EventTableTriggerIO 10058: Operator=0, IOValue=[1], IRC5Controller=? -1, SignalSource=SimulationProject 3637
EventTableTriggerIO 10059: Operator=0, IOValue=[0], IRC5Controller=? -1, SignalSource=SimulationProject 3637
EventTableTriggerIO 10060: Operator=0, IOValue=[0], IRC5Controller=? -1, SignalSource=SimulationProject 3637
EventTableTriggerIO 10061: Operator=0, IOValue=[0], IRC5Controller=? -1, SignalSource=SimulationProject 3637
EventTableTriggerIO 10062: Operator=0, IOValue=[1], IRC5Controller=? -1, SignalSource=SimulationProject 3637
EventTableTriggerIO 10063: Operator=0, IOValue=[1], IRC5Controller=? -1, SignalSource=SimulationProject 3637
EventTableTriggerIO 10064: Operator=0, IOValue=[1], IRC5Controller=? -1, SignalSource=SimulationProject 3637
EventTableTriggerIO 10065: Operator=0, IOValue=[0], IRC5Controller=? -1, SignalSource=SimulationProject 3637
EventTableTriggerIO 10066: Operator=0, IOValue=[0], IRC5Controller=? -1, SignalSource=SimulationProject 3637
EventTableTriggerIO 10067: Operator=0, IOValue=[0], IRC5Controller=? -1, SignalSource=SimulationProject 3637
EventTableTriggerIO 10068: Operator=0, IOValue=[1], IRC5Controller=? -1, SignalSource=SimulationProject 3637
EventTableTriggerIO 10069: Operator=0, IOValue=[1], IRC5Controller=? -1, SignalSource=SimulationProject 3637
EventTableTriggerIO 10070: Operator=0, IOValue=[1], IRC5Controller=? -1, SignalSource=SimulationProject 3637
EventTableTriggerIO 10071: Operator=0, IOValue=[0], IRC5Controller=? -1, SignalSource=SimulationProject 3637
EventTableTriggerIO 10072: Operator=0, IOValue=[0], IRC5Controller=? -1, SignalSource=SimulationProject 3637
EventTableTriggerIO 10073: Operator=0, IOValue=[0], IRC5Controller=? -1, SignalSource=SimulationProject 3637
EventTableTriggerIO 10074: Operator=0, IOValue=[1], IRC5Controller=? -1, SignalSource=SimulationProject 3637
EventTableTriggerIO 10075: Operator=0, IOValue=[1], IRC5Controller=? -1, SignalSource=SimulationProject 3637
EventTableTriggerIO 10076: Operator=0, IOValue=[1], IRC5Controller=? -1, SignalSource=SimulationProject 3637
EventTableTriggerIO 10077: Operator=0, IOValue=[0], IRC5Controller=? -1, SignalSource=SimulationProject 3637
EventTableTriggerIO 10078: Operator=0, IOValue=[0], IRC5Controller=? -1, SignalSource=SimulationProject 3637
EventTableTriggerIO 10079: Operator=0, IOValue=[0], IRC5Controller=? -1, SignalSource=SimulationProject 3637
EventTableTriggerIO 10087: Operator=0, IOValue=[1], IRC5Controller=? -1, SignalSource=SimulationProject 3637
EventTableTriggerIO 10088: Operator=0, IOValue=[0], IRC5Controller=? -1, SignalSource=SimulationProject 3637
EventTableTriggerIO 10089: Operator=0, IOValue=[1], IRC5Controller=? -1, SignalSource=SimulationProject 3637
EventTableTriggerIO 10090: Operator=0, IOValue=[0], IRC5Controller=? -1, SignalSource=SimulationProject 3637
EventTableTriggerIO 10091: Operator=0, IOValue=[1], IRC5Controller=? -1, SignalSource=SimulationProject 3637
EventTableTriggerIO 10092: Operator=0, IOValue=[0], IRC5Controller=? -1, SignalSource=SimulationProject 3637
EventTableTriggerIO 10093: Operator=0, IOValue=[1], IRC5Controller=? -1, SignalSource=SimulationProject 3637
EventTableTriggerIO 10094: Operator=0, IOValue=[0], IRC5Controller=? -1, SignalSource=SimulationProject 3637
EventTableTriggerIO 10095: Operator=0, IOValue=[1], IRC5Controller=? -1, SignalSource=SimulationProject 3637
EventTableTriggerIO 10096: Operator=0, IOValue=[0], IRC5Controller=? -1, SignalSource=SimulationProject 3637
EventTableTriggerIO 10097: Operator=0, IOValue=[1], IRC5Controller=? -1, SignalSource=SimulationProject 3637
EventTableTriggerIO 10098: Operator=0, IOValue=[0], IRC5Controller=? -1, SignalSource=SimulationProject 3637
EventTableTriggerIO 10099: Operator=0, IOValue=[1], IRC5Controller=? -1, SignalSource=SimulationProject 3637
EventTableTriggerIO 10100: Operator=0, IOValue=[0], IRC5Controller=? -1, SignalSource=SimulationProject 3637
EventTableTriggerIO 10101: Operator=0, IOValue=[1], IRC5Controller=? -1, SignalSource=SimulationProject 3637
EventTableTriggerIO 10102: Operator=0, IOValue=[0], IRC5Controller=? -1, SignalSource=SimulationProject 3637
EventTableTriggerIO 10103: Operator=0, IOValue=[1], IRC5Controller=? -1, SignalSource=SimulationProject 3637
EventTableTriggerIO 10104: Operator=0, IOValue=[0], IRC5Controller=? -1, SignalSource=SimulationProject 3637
EventTableTriggerIO 10105: Operator=0, IOValue=[1], IRC5Controller=? -1, SignalSource=SimulationProject 3637
EventTableTriggerIO 10106: Operator=0, IOValue=[0], IRC5Controller=? -1, SignalSource=SimulationProject 3637
EventTableTriggerIO 10107: Operator=0, IOValue=[1], IRC5Controller=? -1, SignalSource=SimulationProject 3637
EventTableTriggerIO 10108: Operator=0, IOValue=[0], IRC5Controller=? -1, SignalSource=SimulationProject 3637
EventTableTriggerIO 10109: Operator=0, IOValue=[1], IRC5Controller=? -1, SignalSource=SimulationProject 3637
EventTableTriggerIO 10110: Operator=0, IOValue=[0], IRC5Controller=? -1, SignalSource=SimulationProject 3637
EventTableTriggerIO 10194: Operator=0, IOValue=[1], IRC5Controller=? -1, SignalSource=SimulationProject 3637
EventTableTriggerIO 10195: Operator=0, IOValue=[1], IRC5Controller=? -1, SignalSource=SimulationProject 3637
EventTableTriggerIO 10196: Operator=0, IOValue=[0], IRC5Controller=? -1, SignalSource=SimulationProject 3637
EventTableTriggerIO 10197: Operator=0, IOValue=[0], IRC5Controller=? -1, SignalSource=SimulationProject 3637
EventTableTriggerIO 10198: Operator=0, IOValue=[1], IRC5Controller=? -1, SignalSource=SimulationProject 3637
EventTableTriggerIO 10199: Operator=0, IOValue=[1], IRC5Controller=? -1, SignalSource=SimulationProject 3637
EventTableTriggerIO 10200: Operator=0, IOValue=[0], IRC5Controller=? -1, SignalSource=SimulationProject 3637
EventTableTriggerIO 10201: Operator=0, IOValue=[0], IRC5Controller=? -1, SignalSource=SimulationProject 3637
EventTableTriggerIO 10202: Operator=0, IOValue=[1], IRC5Controller=? -1, SignalSource=SimulationProject 3637
EventTableTriggerIO 10203: Operator=0, IOValue=[1], IRC5Controller=? -1, SignalSource=SimulationProject 3637
EventTableTriggerIO 10204: Operator=0, IOValue=[0], IRC5Controller=? -1, SignalSource=SimulationProject 3637
EventTableTriggerIO 10205: Operator=0, IOValue=[0], IRC5Controller=? -1, SignalSource=SimulationProject 3637
EventTableTriggerIO 10206: Operator=0, IOValue=[1], IRC5Controller=? -1, SignalSource=SimulationProject 3637
EventTableTriggerIO 10207: Operator=0, IOValue=[1], IRC5Controller=? -1, SignalSource=SimulationProject 3637
EventTableTriggerIO 10208: Operator=0, IOValue=[0], IRC5Controller=? -1, SignalSource=SimulationProject 3637
EventTableTriggerIO 10209: Operator=0, IOValue=[0], IRC5Controller=? -1, SignalSource=SimulationProject 3637
EventTableTriggerIO 10210: Operator=0, IOValue=[1], IRC5Controller=? -1, SignalSource=SimulationProject 3637
EventTableTriggerIO 10211: Operator=0, IOValue=[1], IRC5Controller=? -1, SignalSource=SimulationProject 3637
EventTableTriggerIO 10212: Operator=0, IOValue=[0], IRC5Controller=? -1, SignalSource=SimulationProject 3637
EventTableTriggerIO 10213: Operator=0, IOValue=[0], IRC5Controller=? -1, SignalSource=SimulationProject 3637
EventTableTriggerIO 10214: Operator=0, IOValue=[1], IRC5Controller=? -1, SignalSource=SimulationProject 3637
EventTableTriggerIO 10215: Operator=0, IOValue=[1], IRC5Controller=? -1, SignalSource=SimulationProject 3637
EventTableTriggerIO 10216: Operator=0, IOValue=[0], IRC5Controller=? -1, SignalSource=SimulationProject 3637
EventTableTriggerIO 10217: Operator=0, IOValue=[0], IRC5Controller=? -1, SignalSource=SimulationProject 3637
EventTableTriggerIO 10218: Operator=0, IOValue=[1], IRC5Controller=? -1, SignalSource=SimulationProject 3637
EventTableTriggerIO 10219: Operator=0, IOValue=[1], IRC5Controller=? -1, SignalSource=SimulationProject 3637
EventTableTriggerIO 10220: Operator=0, IOValue=[0], IRC5Controller=? -1, SignalSource=SimulationProject 3637
EventTableTriggerIO 10221: Operator=0, IOValue=[0], IRC5Controller=? -1, SignalSource=SimulationProject 3637
EventTableTriggerIO 10222: Operator=0, IOValue=[1], IRC5Controller=? -1, SignalSource=SimulationProject 3637
EventTableTriggerIO 10223: Operator=0, IOValue=[1], IRC5Controller=? -1, SignalSource=SimulationProject 3637
EventTableTriggerIO 10224: Operator=0, IOValue=[0], IRC5Controller=? -1, SignalSource=SimulationProject 3637
EventTableTriggerIO 10225: Operator=0, IOValue=[0], IRC5Controller=? -1, SignalSource=SimulationProject 3637
EventTableTriggerIO 10226: Operator=0, IOValue=[1], IRC5Controller=? -1, SignalSource=SimulationProject 3637
EventTableTriggerIO 10227: Operator=0, IOValue=[1], IRC5Controller=? -1, SignalSource=SimulationProject 3637
EventTableTriggerIO 10228: Operator=0, IOValue=[0], IRC5Controller=? -1, SignalSource=SimulationProject 3637
EventTableTriggerIO 10229: Operator=0, IOValue=[0], IRC5Controller=? -1, SignalSource=SimulationProject 3637
EventTableTriggerIO 10230: Operator=0, IOValue=[1], IRC5Controller=? -1, SignalSource=SimulationProject 3637
EventTableTriggerIO 10231: Operator=0, IOValue=[1], IRC5Controller=? -1, SignalSource=SimulationProject 3637
EventTableTriggerIO 10232: Operator=0, IOValue=[0], IRC5Controller=? -1, SignalSource=SimulationProject 3637
EventTableTriggerIO 10233: Operator=0, IOValue=[0], IRC5Controller=? -1, SignalSource=SimulationProject 3637
EventTableTriggerIO 10234: Operator=0, IOValue=[1], IRC5Controller=? -1, SignalSource=SimulationProject 3637
EventTableTriggerIO 10235: Operator=0, IOValue=[1], IRC5Controller=? -1, SignalSource=SimulationProject 3637
EventTableTriggerIO 10236: Operator=0, IOValue=[0], IRC5Controller=? -1, SignalSource=SimulationProject 3637
EventTableTriggerIO 10237: Operator=0, IOValue=[0], IRC5Controller=? -1, SignalSource=SimulationProject 3637
EventTableTriggerIO 10238: Operator=0, IOValue=[1], IRC5Controller=? -1, SignalSource=SimulationProject 3637
EventTableTriggerIO 10239: Operator=0, IOValue=[1], IRC5Controller=? -1, SignalSource=SimulationProject 3637
EventTableTriggerIO 10240: Operator=0, IOValue=[0], IRC5Controller=? -1, SignalSource=SimulationProject 3637
EventTableTriggerIO 10241: Operator=0, IOValue=[0], IRC5Controller=? -1, SignalSource=SimulationProject 3637
EventTableEntry 10242: ActivationMode=2, Cyclic=false, Group=, Trigger=doAxelTool_L 10243, Actions=[EventTableActionAttach 10244], Comment=
EventTableTriggerIO 10243: Operator=0, IOValue=[1], IRC5Controller=? -1, SignalSource=SimulationProject 3637
EventTableActionAttach 10244: MountObject=false, FlangeIndext=0, FindNearest=false, AttachmentParent=IRB6660_100_335__01_L 3595, AttachmentChild=AxelPinTool_L 5996, Offset=[X=1, Y=0, Z=0, W=0, X=0, Y=1, Z=0, W=0, X=0, Y=0, Z=1, W=0, X=0, Y=0, Z=0, W=1]
EventTableTriggerIO 10245: Operator=0, IOValue=[1], IRC5Controller=? -1, SignalSource=SimulationProject 3637
EventTableEntry 10246: ActivationMode=2, Cyclic=false, Group=, Trigger=doAxelTool_L 10247, Actions=[EventTableActionDetach 10248], Comment=
EventTableTriggerIO 10247: Operator=0, IOValue=[0], IRC5Controller=? -1, SignalSource=SimulationProject 3637
EventTableActionDetach 10248: AttachmentParent=IRB6660_100_335__01_L 3595, AttachmentChild=AxelPinTool_L 5996
EventTableTriggerIO 10249: Operator=0, IOValue=[0], IRC5Controller=? -1, SignalSource=SimulationProject 3637
EventTableEntry 10250: ActivationMode=2, Cyclic=false, Group=, Trigger=doAxel_L 10251, Actions=[EventTableActionAttach 10252], Comment=
EventTableTriggerIO 10251: Operator=0, IOValue=[1], IRC5Controller=? -1, SignalSource=SimulationProject 3637
EventTableActionAttach 10252: MountObject=false, FlangeIndext=0, FindNearest=true, AttachmentParent=AxelPinTool_L 5996, AttachmentChild=? -1, Offset=[X=1, Y=0, Z=0, W=0, X=0, Y=1, Z=0, W=0, X=0, Y=0, Z=1, W=0, X=0, Y=0, Z=0, W=1]
EventTableTriggerIO 10253: Operator=0, IOValue=[1], IRC5Controller=? -1, SignalSource=SimulationProject 3637
EventTableEntry 10254: ActivationMode=2, Cyclic=false, Group=, Trigger=doAxel_L 10255, Actions=[EventTableActionDetach 10256], Comment=
EventTableTriggerIO 10255: Operator=0, IOValue=[0], IRC5Controller=? -1, SignalSource=SimulationProject 3637
EventTableActionDetach 10256: AttachmentParent=AxelPinTool_L 5996, AttachmentChild=? -1
EventTableTriggerIO 10257: Operator=0, IOValue=[0], IRC5Controller=? -1, SignalSource=SimulationProject 3637
EventTableTriggerIO 10629: Operator=0, IOValue=[1], IRC5Controller=? -1, SignalSource=SimulationProject 3637
EventTableTriggerIO 10630: Operator=0, IOValue=[0], IRC5Controller=? -1, SignalSource=SimulationProject 3637
EventTableTriggerIO 10631: Operator=0, IOValue=[1], IRC5Controller=? -1, SignalSource=SimulationProject 3637
EventTableTriggerIO 10632: Operator=0, IOValue=[0], IRC5Controller=? -1, SignalSource=SimulationProject 3637
EventTableTriggerIO 10633: Operator=0, IOValue=[1], IRC5Controller=? -1, SignalSource=SimulationProject 3637
EventTableTriggerIO 10634: Operator=0, IOValue=[0], IRC5Controller=? -1, SignalSource=SimulationProject 3637
EventTableTriggerIO 10635: Operator=0, IOValue=[1], IRC5Controller=? -1, SignalSource=SimulationProject 3637
EventTableTriggerIO 10636: Operator=0, IOValue=[0], IRC5Controller=? -1, SignalSource=SimulationProject 3637
EventTableTriggerIO 10637: Operator=0, IOValue=[1], IRC5Controller=? -1, SignalSource=SimulationProject 3637
EventTableTriggerIO 10638: Operator=0, IOValue=[0], IRC5Controller=? -1, SignalSource=SimulationProject 3637
EventTableTriggerIO 10639: Operator=0, IOValue=[1], IRC5Controller=? -1, SignalSource=SimulationProject 3637
EventTableTriggerIO 10640: Operator=0, IOValue=[0], IRC5Controller=? -1, SignalSource=SimulationProject 3637
EventTableTriggerIO 10641: Operator=0, IOValue=[1], IRC5Controller=? -1, SignalSource=SimulationProject 3637
EventTableTriggerIO 10642: Operator=0, IOValue=[0], IRC5Controller=? -1, SignalSource=SimulationProject 3637
EventTableTriggerIO 10643: Operator=0, IOValue=[1], IRC5Controller=? -1, SignalSource=SimulationProject 3637
EventTableTriggerIO 10644: Operator=0, IOValue=[0], IRC5Controller=? -1, SignalSource=SimulationProject 3637
EventTableTriggerIO 10645: Operator=0, IOValue=[1], IRC5Controller=? -1, SignalSource=SimulationProject 3637
EventTableTriggerIO 10646: Operator=0, IOValue=[0], IRC5Controller=? -1, SignalSource=SimulationProject 3637
EventTableTriggerIO 10647: Operator=0, IOValue=[1], IRC5Controller=? -1, SignalSource=SimulationProject 3637
EventTableTriggerIO 10648: Operator=0, IOValue=[0], IRC5Controller=? -1, SignalSource=SimulationProject 3637
EventTableTriggerIO 10649: Operator=0, IOValue=[1], IRC5Controller=? -1, SignalSource=SimulationProject 3637
EventTableTriggerIO 10650: Operator=0, IOValue=[0], IRC5Controller=? -1, SignalSource=SimulationProject 3637
EventTableTriggerIO 10651: Operator=0, IOValue=[1], IRC5Controller=? -1, SignalSource=SimulationProject 3637
EventTableTriggerIO 10652: Operator=0, IOValue=[0], IRC5Controller=? -1, SignalSource=SimulationProject 3637
EventTableTriggerIO 10653: Operator=0, IOValue=[1], IRC5Controller=? -1, SignalSource=SimulationProject 3637
EventTableTriggerIO 10654: Operator=0, IOValue=[0], IRC5Controller=? -1, SignalSource=SimulationProject 3637
EventTableTriggerIO 10655: Operator=0, IOValue=[1], IRC5Controller=? -1, SignalSource=SimulationProject 3637
EventTableTriggerIO 10656: Operator=0, IOValue=[0], IRC5Controller=? -1, SignalSource=SimulationProject 3637
EventTableTriggerIO 10664: Operator=0, IOValue=[1], IRC5Controller=? -1, SignalSource=SimulationProject 3637
EventTableTriggerIO 10665: Operator=0, IOValue=[0], IRC5Controller=? -1, SignalSource=SimulationProject 3637
EventTableTriggerIO 10666: Operator=0, IOValue=[1], IRC5Controller=? -1, SignalSource=SimulationProject 3637
EventTableTriggerIO 10667: Operator=0, IOValue=[0], IRC5Controller=? -1, SignalSource=SimulationProject 3637
EventTableTriggerIO 10668: Operator=0, IOValue=[1], IRC5Controller=? -1, SignalSource=SimulationProject 3637
EventTableTriggerIO 10669: Operator=0, IOValue=[0], IRC5Controller=? -1, SignalSource=SimulationProject 3637
EventTableTriggerIO 10670: Operator=0, IOValue=[1], IRC5Controller=? -1, SignalSource=SimulationProject 3637
EventTableTriggerIO 10671: Operator=0, IOValue=[0], IRC5Controller=? -1, SignalSource=SimulationProject 3637
EventTableTriggerIO 10672: Operator=0, IOValue=[1], IRC5Controller=? -1, SignalSource=SimulationProject 3637
EventTableTriggerIO 10673: Operator=0, IOValue=[0], IRC5Controller=? -1, SignalSource=SimulationProject 3637
EventTableTriggerIO 10674: Operator=0, IOValue=[1], IRC5Controller=? -1, SignalSource=SimulationProject 3637
EventTableTriggerIO 10675: Operator=0, IOValue=[0], IRC5Controller=? -1, SignalSource=SimulationProject 3637
EventTableTriggerIO 10676: Operator=0, IOValue=[1], IRC5Controller=? -1, SignalSource=SimulationProject 3637
EventTableTriggerIO 10677: Operator=0, IOValue=[0], IRC5Controller=? -1, SignalSource=SimulationProject 3637
EventTableTriggerIO 10678: Operator=0, IOValue=[1], IRC5Controller=? -1, SignalSource=SimulationProject 3637
EventTableTriggerIO 10679: Operator=0, IOValue=[0], IRC5Controller=? -1, SignalSource=SimulationProject 3637
EventTableTriggerIO 10680: Operator=0, IOValue=[1], IRC5Controller=? -1, SignalSource=SimulationProject 3637
EventTableTriggerIO 10681: Operator=0, IOValue=[0], IRC5Controller=? -1, SignalSource=SimulationProject 3637
EventTableTriggerIO 10682: Operator=0, IOValue=[1], IRC5Controller=? -1, SignalSource=SimulationProject 3637
EventTableTriggerIO 10683: Operator=0, IOValue=[0], IRC5Controller=? -1, SignalSource=SimulationProject 3637
EventTableTriggerIO 10684: Operator=0, IOValue=[1], IRC5Controller=? -1, SignalSource=SimulationProject 3637
EventTableTriggerIO 10685: Operator=0, IOValue=[0], IRC5Controller=? -1, SignalSource=SimulationProject 3637
EventTableTriggerIO 10686: Operator=0, IOValue=[1], IRC5Controller=? -1, SignalSource=SimulationProject 3637
EventTableTriggerIO 10687: Operator=0, IOValue=[0], IRC5Controller=? -1, SignalSource=SimulationProject 3637
EventTableTriggerIO 10688: Operator=0, IOValue=[1], IRC5Controller=? -1, SignalSource=SimulationProject 3637
EventTableTriggerIO 10689: Operator=0, IOValue=[0], IRC5Controller=? -1, SignalSource=SimulationProject 3637
EventTableTriggerIO 10690: Operator=0, IOValue=[1], IRC5Controller=? -1, SignalSource=SimulationProject 3637
EventTableTriggerIO 10691: Operator=0, IOValue=[0], IRC5Controller=? -1, SignalSource=SimulationProject 3637
EventTableTriggerIO 10748: Operator=0, IOValue=[1], IRC5Controller=? -1, SignalSource=SimulationProject 3637
EventTableTriggerIO 10749: Operator=0, IOValue=[1], IRC5Controller=? -1, SignalSource=SimulationProject 3637
EventTableTriggerIO 10750: Operator=0, IOValue=[1], IRC5Controller=? -1, SignalSource=SimulationProject 3637
EventTableTriggerIO 10751: Operator=0, IOValue=[0], IRC5Controller=? -1, SignalSource=SimulationProject 3637
EventTableTriggerIO 10752: Operator=0, IOValue=[0], IRC5Controller=? -1, SignalSource=SimulationProject 3637
EventTableTriggerIO 10753: Operator=0, IOValue=[0], IRC5Controller=? -1, SignalSource=SimulationProject 3637
EventTableTriggerIO 10754: Operator=0, IOValue=[1], IRC5Controller=? -1, SignalSource=SimulationProject 3637
EventTableTriggerIO 10755: Operator=0, IOValue=[1], IRC5Controller=? -1, SignalSource=SimulationProject 3637
EventTableTriggerIO 10756: Operator=0, IOValue=[1], IRC5Controller=? -1, SignalSource=SimulationProject 3637
EventTableTriggerIO 10757: Operator=0, IOValue=[0], IRC5Controller=? -1, SignalSource=SimulationProject 3637
EventTableTriggerIO 10758: Operator=0, IOValue=[0], IRC5Controller=? -1, SignalSource=SimulationProject 3637
EventTableTriggerIO 10759: Operator=0, IOValue=[0], IRC5Controller=? -1, SignalSource=SimulationProject 3637
EventTableTriggerIO 10760: Operator=0, IOValue=[1], IRC5Controller=? -1, SignalSource=SimulationProject 3637
EventTableTriggerIO 10761: Operator=0, IOValue=[1], IRC5Controller=? -1, SignalSource=SimulationProject 3637
EventTableTriggerIO 10762: Operator=0, IOValue=[1], IRC5Controller=? -1, SignalSource=SimulationProject 3637
EventTableTriggerIO 10763: Operator=0, IOValue=[0], IRC5Controller=? -1, SignalSource=SimulationProject 3637
EventTableTriggerIO 10764: Operator=0, IOValue=[0], IRC5Controller=? -1, SignalSource=SimulationProject 3637
EventTableTriggerIO 10765: Operator=0, IOValue=[0], IRC5Controller=? -1, SignalSource=SimulationProject 3637
EventTableTriggerIO 10766: Operator=0, IOValue=[1], IRC5Controller=? -1, SignalSource=SimulationProject 3637
EventTableTriggerIO 10767: Operator=0, IOValue=[1], IRC5Controller=? -1, SignalSource=SimulationProject 3637
EventTableTriggerIO 10768: Operator=0, IOValue=[1], IRC5Controller=? -1, SignalSource=SimulationProject 3637
EventTableTriggerIO 10769: Operator=0, IOValue=[0], IRC5Controller=? -1, SignalSource=SimulationProject 3637
EventTableTriggerIO 10770: Operator=0, IOValue=[0], IRC5Controller=? -1, SignalSource=SimulationProject 3637
EventTableTriggerIO 10771: Operator=0, IOValue=[0], IRC5Controller=? -1, SignalSource=SimulationProject 3637
EventTableTriggerIO 10772: Operator=0, IOValue=[1], IRC5Controller=? -1, SignalSource=SimulationProject 3637
EventTableTriggerIO 10773: Operator=0, IOValue=[1], IRC5Controller=? -1, SignalSource=SimulationProject 3637
EventTableTriggerIO 10774: Operator=0, IOValue=[1], IRC5Controller=? -1, SignalSource=SimulationProject 3637
EventTableTriggerIO 10775: Operator=0, IOValue=[0], IRC5Controller=? -1, SignalSource=SimulationProject 3637
EventTableTriggerIO 10776: Operator=0, IOValue=[0], IRC5Controller=? -1, SignalSource=SimulationProject 3637
EventTableTriggerIO 10777: Operator=0, IOValue=[0], IRC5Controller=? -1, SignalSource=SimulationProject 3637
EventTableTriggerIO 10778: Operator=0, IOValue=[1], IRC5Controller=? -1, SignalSource=SimulationProject 3637
EventTableTriggerIO 10779: Operator=0, IOValue=[1], IRC5Controller=? -1, SignalSource=SimulationProject 3637
EventTableTriggerIO 10780: Operator=0, IOValue=[1], IRC5Controller=? -1, SignalSource=SimulationProject 3637
EventTableTriggerIO 10781: Operator=0, IOValue=[0], IRC5Controller=? -1, SignalSource=SimulationProject 3637
EventTableTriggerIO 10782: Operator=0, IOValue=[0], IRC5Controller=? -1, SignalSource=SimulationProject 3637
EventTableTriggerIO 10783: Operator=0, IOValue=[0], IRC5Controller=? -1, SignalSource=SimulationProject 3637
EventTableTriggerIO 10784: Operator=0, IOValue=[1], IRC5Controller=? -1, SignalSource=SimulationProject 3637
EventTableTriggerIO 10785: Operator=0, IOValue=[1], IRC5Controller=? -1, SignalSource=SimulationProject 3637
EventTableTriggerIO 10786: Operator=0, IOValue=[1], IRC5Controller=? -1, SignalSource=SimulationProject 3637
EventTableTriggerIO 10787: Operator=0, IOValue=[0], IRC5Controller=? -1, SignalSource=SimulationProject 3637
EventTableTriggerIO 10788: Operator=0, IOValue=[0], IRC5Controller=? -1, SignalSource=SimulationProject 3637
EventTableTriggerIO 10789: Operator=0, IOValue=[0], IRC5Controller=? -1, SignalSource=SimulationProject 3637
EventTableTriggerIO 10790: Operator=0, IOValue=[1], IRC5Controller=? -1, SignalSource=SimulationProject 3637
EventTableTriggerIO 10791: Operator=0, IOValue=[1], IRC5Controller=? -1, SignalSource=SimulationProject 3637
EventTableTriggerIO 10792: Operator=0, IOValue=[1], IRC5Controller=? -1, SignalSource=SimulationProject 3637
EventTableTriggerIO 10793: Operator=0, IOValue=[0], IRC5Controller=? -1, SignalSource=SimulationProject 3637
EventTableTriggerIO 10794: Operator=0, IOValue=[0], IRC5Controller=? -1, SignalSource=SimulationProject 3637
EventTableTriggerIO 10795: Operator=0, IOValue=[0], IRC5Controller=? -1, SignalSource=SimulationProject 3637
EventTableTriggerIO 10796: Operator=0, IOValue=[1], IRC5Controller=? -1, SignalSource=SimulationProject 3637
EventTableTriggerIO 10797: Operator=0, IOValue=[1], IRC5Controller=? -1, SignalSource=SimulationProject 3637
EventTableTriggerIO 10798: Operator=0, IOValue=[1], IRC5Controller=? -1, SignalSource=SimulationProject 3637
EventTableTriggerIO 10799: Operator=0, IOValue=[0], IRC5Controller=? -1, SignalSource=SimulationProject 3637
EventTableTriggerIO 10800: Operator=0, IOValue=[0], IRC5Controller=? -1, SignalSource=SimulationProject 3637
EventTableTriggerIO 10801: Operator=0, IOValue=[0], IRC5Controller=? -1, SignalSource=SimulationProject 3637
EventTableTriggerIO 10802: Operator=0, IOValue=[1], IRC5Controller=? -1, SignalSource=SimulationProject 3637
EventTableTriggerIO 10803: Operator=0, IOValue=[1], IRC5Controller=? -1, SignalSource=SimulationProject 3637
EventTableTriggerIO 10804: Operator=0, IOValue=[1], IRC5Controller=? -1, SignalSource=SimulationProject 3637
EventTableTriggerIO 10805: Operator=0, IOValue=[0], IRC5Controller=? -1, SignalSource=SimulationProject 3637
EventTableTriggerIO 10806: Operator=0, IOValue=[0], IRC5Controller=? -1, SignalSource=SimulationProject 3637
EventTableTriggerIO 10807: Operator=0, IOValue=[0], IRC5Controller=? -1, SignalSource=SimulationProject 3637
EventTableTriggerIO 10808: Operator=0, IOValue=[1], IRC5Controller=? -1, SignalSource=SimulationProject 3637
EventTableTriggerIO 10809: Operator=0, IOValue=[1], IRC5Controller=? -1, SignalSource=SimulationProject 3637
EventTableTriggerIO 10810: Operator=0, IOValue=[1], IRC5Controller=? -1, SignalSource=SimulationProject 3637
EventTableTriggerIO 10811: Operator=0, IOValue=[0], IRC5Controller=? -1, SignalSource=SimulationProject 3637
EventTableTriggerIO 10812: Operator=0, IOValue=[0], IRC5Controller=? -1, SignalSource=SimulationProject 3637
EventTableTriggerIO 10813: Operator=0, IOValue=[0], IRC5Controller=? -1, SignalSource=SimulationProject 3637
EventTableTriggerIO 10814: Operator=0, IOValue=[1], IRC5Controller=? -1, SignalSource=SimulationProject 3637
EventTableTriggerIO 10815: Operator=0, IOValue=[1], IRC5Controller=? -1, SignalSource=SimulationProject 3637
EventTableTriggerIO 10816: Operator=0, IOValue=[1], IRC5Controller=? -1, SignalSource=SimulationProject 3637
EventTableTriggerIO 10817: Operator=0, IOValue=[0], IRC5Controller=? -1, SignalSource=SimulationProject 3637
EventTableTriggerIO 10818: Operator=0, IOValue=[0], IRC5Controller=? -1, SignalSource=SimulationProject 3637
EventTableTriggerIO 10819: Operator=0, IOValue=[0], IRC5Controller=? -1, SignalSource=SimulationProject 3637
EventTableTriggerIO 10820: Operator=0, IOValue=[1], IRC5Controller=? -1, SignalSource=SimulationProject 3637
EventTableTriggerIO 10821: Operator=0, IOValue=[1], IRC5Controller=? -1, SignalSource=SimulationProject 3637
EventTableTriggerIO 10822: Operator=0, IOValue=[1], IRC5Controller=? -1, SignalSource=SimulationProject 3637
EventTableTriggerIO 10823: Operator=0, IOValue=[0], IRC5Controller=? -1, SignalSource=SimulationProject 3637
EventTableTriggerIO 10824: Operator=0, IOValue=[0], IRC5Controller=? -1, SignalSource=SimulationProject 3637
EventTableTriggerIO 10825: Operator=0, IOValue=[0], IRC5Controller=? -1, SignalSource=SimulationProject 3637
EventTableTriggerIO 10826: Operator=0, IOValue=[1], IRC5Controller=? -1, SignalSource=SimulationProject 3637
EventTableTriggerIO 10827: Operator=0, IOValue=[1], IRC5Controller=? -1, SignalSource=SimulationProject 3637
EventTableTriggerIO 10828: Operator=0, IOValue=[1], IRC5Controller=? -1, SignalSource=SimulationProject 3637
EventTableTriggerIO 10829: Operator=0, IOValue=[0], IRC5Controller=? -1, SignalSource=SimulationProject 3637
EventTableTriggerIO 10830: Operator=0, IOValue=[0], IRC5Controller=? -1, SignalSource=SimulationProject 3637
EventTableTriggerIO 10831: Operator=0, IOValue=[0], IRC5Controller=? -1, SignalSource=SimulationProject 3637
EventTableTriggerIO 11467: Operator=0, IOValue=[1], IRC5Controller=? -1, SignalSource=SimulationProject 3637
EventTableTriggerIO 11468: Operator=0, IOValue=[1], IRC5Controller=? -1, SignalSource=SimulationProject 3637
EventTableTriggerIO 11469: Operator=0, IOValue=[0], IRC5Controller=? -1, SignalSource=SimulationProject 3637
EventTableTriggerIO 11470: Operator=0, IOValue=[0], IRC5Controller=? -1, SignalSource=SimulationProject 3637
EventTableTriggerIO 11471: Operator=0, IOValue=[1], IRC5Controller=? -1, SignalSource=SimulationProject 3637
EventTableTriggerIO 11472: Operator=0, IOValue=[1], IRC5Controller=? -1, SignalSource=SimulationProject 3637
EventTableTriggerIO 11473: Operator=0, IOValue=[0], IRC5Controller=? -1, SignalSource=SimulationProject 3637
EventTableTriggerIO 11474: Operator=0, IOValue=[0], IRC5Controller=? -1, SignalSource=SimulationProject 3637
EventTableTriggerIO 11475: Operator=0, IOValue=[1], IRC5Controller=? -1, SignalSource=SimulationProject 3637
EventTableTriggerIO 11476: Operator=0, IOValue=[1], IRC5Controller=? -1, SignalSource=SimulationProject 3637
EventTableTriggerIO 11477: Operator=0, IOValue=[0], IRC5Controller=? -1, SignalSource=SimulationProject 3637
EventTableTriggerIO 11478: Operator=0, IOValue=[0], IRC5Controller=? -1, SignalSource=SimulationProject 3637
EventTableTriggerIO 11479: Operator=0, IOValue=[1], IRC5Controller=? -1, SignalSource=SimulationProject 3637
EventTableTriggerIO 11480: Operator=0, IOValue=[1], IRC5Controller=? -1, SignalSource=SimulationProject 3637
EventTableTriggerIO 11481: Operator=0, IOValue=[0], IRC5Controller=? -1, SignalSource=SimulationProject 3637
EventTableTriggerIO 11482: Operator=0, IOValue=[0], IRC5Controller=? -1, SignalSource=SimulationProject 3637
EventTableTriggerIO 11483: Operator=0, IOValue=[1], IRC5Controller=? -1, SignalSource=SimulationProject 3637
EventTableTriggerIO 11484: Operator=0, IOValue=[1], IRC5Controller=? -1, SignalSource=SimulationProject 3637
EventTableTriggerIO 11485: Operator=0, IOValue=[0], IRC5Controller=? -1, SignalSource=SimulationProject 3637
EventTableTriggerIO 11486: Operator=0, IOValue=[0], IRC5Controller=? -1, SignalSource=SimulationProject 3637
EventTableTriggerIO 11487: Operator=0, IOValue=[1], IRC5Controller=? -1, SignalSource=SimulationProject 3637
EventTableTriggerIO 11488: Operator=0, IOValue=[1], IRC5Controller=? -1, SignalSource=SimulationProject 3637
EventTableTriggerIO 11489: Operator=0, IOValue=[0], IRC5Controller=? -1, SignalSource=SimulationProject 3637
EventTableTriggerIO 11490: Operator=0, IOValue=[0], IRC5Controller=? -1, SignalSource=SimulationProject 3637
EventTableTriggerIO 11491: Operator=0, IOValue=[1], IRC5Controller=? -1, SignalSource=SimulationProject 3637
EventTableTriggerIO 11492: Operator=0, IOValue=[1], IRC5Controller=? -1, SignalSource=SimulationProject 3637
EventTableTriggerIO 11493: Operator=0, IOValue=[0], IRC5Controller=? -1, SignalSource=SimulationProject 3637
EventTableTriggerIO 11494: Operator=0, IOValue=[0], IRC5Controller=? -1, SignalSource=SimulationProject 3637
EventTableTriggerIO 11495: Operator=0, IOValue=[1], IRC5Controller=? -1, SignalSource=SimulationProject 3637
EventTableTriggerIO 11496: Operator=0, IOValue=[1], IRC5Controller=? -1, SignalSource=SimulationProject 3637
EventTableTriggerIO 11497: Operator=0, IOValue=[0], IRC5Controller=? -1, SignalSource=SimulationProject 3637
EventTableTriggerIO 11498: Operator=0, IOValue=[0], IRC5Controller=? -1, SignalSource=SimulationProject 3637
EventTableTriggerIO 11499: Operator=0, IOValue=[1], IRC5Controller=? -1, SignalSource=SimulationProject 3637
EventTableTriggerIO 11500: Operator=0, IOValue=[1], IRC5Controller=? -1, SignalSource=SimulationProject 3637
EventTableTriggerIO 11501: Operator=0, IOValue=[0], IRC5Controller=? -1, SignalSource=SimulationProject 3637
EventTableTriggerIO 11502: Operator=0, IOValue=[0], IRC5Controller=? -1, SignalSource=SimulationProject 3637
EventTableTriggerIO 11503: Operator=0, IOValue=[1], IRC5Controller=? -1, SignalSource=SimulationProject 3637
EventTableTriggerIO 11504: Operator=0, IOValue=[1], IRC5Controller=? -1, SignalSource=SimulationProject 3637
EventTableTriggerIO 11505: Operator=0, IOValue=[0], IRC5Controller=? -1, SignalSource=SimulationProject 3637
EventTableTriggerIO 11506: Operator=0, IOValue=[0], IRC5Controller=? -1, SignalSource=SimulationProject 3637
EventTableTriggerIO 11507: Operator=0, IOValue=[1], IRC5Controller=? -1, SignalSource=SimulationProject 3637
EventTableTriggerIO 11508: Operator=0, IOValue=[1], IRC5Controller=? -1, SignalSource=SimulationProject 3637
EventTableTriggerIO 11509: Operator=0, IOValue=[0], IRC5Controller=? -1, SignalSource=SimulationProject 3637
EventTableTriggerIO 11510: Operator=0, IOValue=[0], IRC5Controller=? -1, SignalSource=SimulationProject 3637
EventTableTriggerIO 11511: Operator=0, IOValue=[1], IRC5Controller=? -1, SignalSource=SimulationProject 3637
EventTableTriggerIO 11512: Operator=0, IOValue=[1], IRC5Controller=? -1, SignalSource=SimulationProject 3637
EventTableTriggerIO 11513: Operator=0, IOValue=[0], IRC5Controller=? -1, SignalSource=SimulationProject 3637
EventTableTriggerIO 11514: Operator=0, IOValue=[0], IRC5Controller=? -1, SignalSource=SimulationProject 3637
EventTableTriggerIO 11515: Operator=0, IOValue=[1], IRC5Controller=? -1, SignalSource=SimulationProject 3637
EventTableTriggerIO 11516: Operator=0, IOValue=[1], IRC5Controller=? -1, SignalSource=SimulationProject 3637
EventTableTriggerIO 11517: Operator=0, IOValue=[0], IRC5Controller=? -1, SignalSource=SimulationProject 3637
EventTableTriggerIO 11518: Operator=0, IOValue=[0], IRC5Controller=? -1, SignalSource=SimulationProject 3637
EventTableTriggerIO 11519: Operator=0, IOValue=[1], IRC5Controller=? -1, SignalSource=SimulationProject 3637
EventTableTriggerIO 11520: Operator=0, IOValue=[1], IRC5Controller=? -1, SignalSource=SimulationProject 3637
EventTableTriggerIO 11521: Operator=0, IOValue=[0], IRC5Controller=? -1, SignalSource=SimulationProject 3637
EventTableTriggerIO 11522: Operator=0, IOValue=[0], IRC5Controller=? -1, SignalSource=SimulationProject 3637
EventTableEntry 11523: ActivationMode=2, Cyclic=false, Group=, Trigger=doLinkTool_L 11524, Actions=[EventTableActionAttach 11525], Comment=
EventTableTriggerIO 11524: Operator=0, IOValue=[1], IRC5Controller=? -1, SignalSource=SimulationProject 3637
EventTableActionAttach 11525: MountObject=false, FlangeIndext=0, FindNearest=false, AttachmentParent=IRB6660_100_335__01_L 3595, AttachmentChild=LinkTool_L 7468, Offset=[X=1, Y=0, Z=0, W=0, X=0, Y=1, Z=0, W=0, X=0, Y=0, Z=1, W=0, X=0, Y=0, Z=0, W=1]
EventTableTriggerIO 11526: Operator=0, IOValue=[1], IRC5Controller=? -1, SignalSource=SimulationProject 3637
EventTableTriggerIO 11527: Operator=0, IOValue=[1], IRC5Controller=? -1, SignalSource=SimulationProject 3637
EventTableEntry 11528: ActivationMode=2, Cyclic=false, Group=, Trigger=doLinkTool_L 11529, Actions=[EventTableActionDetach 11530], Comment=
EventTableTriggerIO 11529: Operator=0, IOValue=[0], IRC5Controller=? -1, SignalSource=SimulationProject 3637
EventTableActionDetach 11530: AttachmentParent=IRB6660_100_335__01_L 3595, AttachmentChild=LinkTool_L 7468
EventTableTriggerIO 11531: Operator=0, IOValue=[0], IRC5Controller=? -1, SignalSource=SimulationProject 3637
EventTableTriggerIO 11532: Operator=0, IOValue=[0], IRC5Controller=? -1, SignalSource=SimulationProject 3637
EventTableEntry 11533: ActivationMode=2, Cyclic=false, Group=, Trigger=doLink_L 11534, Actions=[EventTableActionAttach 11535], Comment=
EventTableTriggerIO 11534: Operator=0, IOValue=[1], IRC5Controller=? -1, SignalSource=SimulationProject 3637
EventTableActionAttach 11535: MountObject=false, FlangeIndext=0, FindNearest=true, AttachmentParent=LinkTool_L 7468, AttachmentChild=? -1, Offset=[X=1, Y=0, Z=0, W=0, X=0, Y=1, Z=0, W=0, X=0, Y=0, Z=1, W=0, X=0, Y=0, Z=0, W=1]
EventTableTriggerIO 11536: Operator=0, IOValue=[1], IRC5Controller=? -1, SignalSource=SimulationProject 3637
EventTableTriggerIO 11537: Operator=0, IOValue=[1], IRC5Controller=? -1, SignalSource=SimulationProject 3637
EventTableEntry 11538: ActivationMode=2, Cyclic=false, Group=, Trigger=doLink_L 11539, Actions=[EventTableActionDetach 11540], Comment=
EventTableTriggerIO 11539: Operator=0, IOValue=[0], IRC5Controller=? -1, SignalSource=SimulationProject 3637
EventTableActionDetach 11540: AttachmentParent=LinkTool_L 7468, AttachmentChild=? -1
EventTableTriggerIO 11541: Operator=0, IOValue=[0], IRC5Controller=? -1, SignalSource=SimulationProject 3637
EventTableTriggerIO 11542: Operator=0, IOValue=[0], IRC5Controller=? -1, SignalSource=SimulationProject 3637
EventTableEntry 11543: ActivationMode=2, Cyclic=false, Group=, Trigger=doArmTool_L 11544, Actions=[EventTableActionAttach 11545], Comment=
EventTableTriggerIO 11544: Operator=0, IOValue=[1], IRC5Controller=? -1, SignalSource=SimulationProject 3637
EventTableActionAttach 11545: MountObject=false, FlangeIndext=0, FindNearest=false, AttachmentParent=IRB6660_100_335__01_L 3595, AttachmentChild=ArmPinTool_L 5999, Offset=[X=1, Y=0, Z=0, W=0, X=0, Y=1, Z=0, W=0, X=0, Y=0, Z=1, W=0, X=0, Y=0, Z=0, W=1]
EventTableTriggerIO 11546: Operator=0, IOValue=[1], IRC5Controller=? -1, SignalSource=SimulationProject 3637
EventTableTriggerIO 11547: Operator=0, IOValue=[1], IRC5Controller=? -1, SignalSource=SimulationProject 3637
EventTableEntry 11548: ActivationMode=2, Cyclic=false, Group=, Trigger=doArmTool_L 11549, Actions=[EventTableActionDetach 11550], Comment=
EventTableTriggerIO 11549: Operator=0, IOValue=[0], IRC5Controller=? -1, SignalSource=SimulationProject 3637
EventTableActionDetach 11550: AttachmentParent=IRB6660_100_335__01_L 3595, AttachmentChild=ArmPinTool_L 5999
EventTableTriggerIO 11551: Operator=0, IOValue=[0], IRC5Controller=? -1, SignalSource=SimulationProject 3637
EventTableTriggerIO 11552: Operator=0, IOValue=[0], IRC5Controller=? -1, SignalSource=SimulationProject 3637
EventTableEntry 11553: ActivationMode=2, Cyclic=false, Group=, Trigger=doArm_L 11554, Actions=[EventTableActionAttach 11555], Comment=
EventTableTriggerIO 11554: Operator=0, IOValue=[1], IRC5Controller=? -1, SignalSource=SimulationProject 3637
EventTableActionAttach 11555: MountObject=false, FlangeIndext=0, FindNearest=true, AttachmentParent=ArmPinTool_L 5999, AttachmentChild=? -1, Offset=[X=1, Y=0, Z=0, W=0, X=0, Y=1, Z=0, W=0, X=0, Y=0, Z=1, W=0, X=0, Y=0, Z=0, W=1]
EventTableTriggerIO 11556: Operator=0, IOValue=[1], IRC5Controller=? -1, SignalSource=SimulationProject 3637
EventTableTriggerIO 11557: Operator=0, IOValue=[1], IRC5Controller=? -1, SignalSource=SimulationProject 3637
EventTableEntry 11558: ActivationMode=2, Cyclic=false, Group=, Trigger=doArm_L 11559, Actions=[EventTableActionDetach 11560], Comment=
EventTableTriggerIO 11559: Operator=0, IOValue=[0], IRC5Controller=? -1, SignalSource=SimulationProject 3637
EventTableActionDetach 11560: AttachmentParent=ArmPinTool_L 5999, AttachmentChild=? -1
EventTableTriggerIO 11561: Operator=0, IOValue=[0], IRC5Controller=? -1, SignalSource=SimulationProject 3637
EventTableTriggerIO 11562: Operator=0, IOValue=[0], IRC5Controller=? -1, SignalSource=SimulationProject 3637
EventTableTriggerIO 11568: Operator=0, IOValue=[1], IRC5Controller=? -1, SignalSource=SimulationProject 3637
EventTableTriggerIO 11569: Operator=0, IOValue=[1], IRC5Controller=? -1, SignalSource=SimulationProject 3637
EventTableTriggerIO 11570: Operator=0, IOValue=[0], IRC5Controller=? -1, SignalSource=SimulationProject 3637
EventTableTriggerIO 11571: Operator=0, IOValue=[0], IRC5Controller=? -1, SignalSource=SimulationProject 3637
EventTableTriggerIO 11572: Operator=0, IOValue=[1], IRC5Controller=? -1, SignalSource=SimulationProject 3637
EventTableTriggerIO 11573: Operator=0, IOValue=[1], IRC5Controller=? -1, SignalSource=SimulationProject 3637
EventTableTriggerIO 11574: Operator=0, IOValue=[0], IRC5Controller=? -1, SignalSource=SimulationProject 3637
EventTableTriggerIO 11575: Operator=0, IOValue=[0], IRC5Controller=? -1, SignalSource=SimulationProject 3637
EventTableTriggerIO 11576: Operator=0, IOValue=[1], IRC5Controller=? -1, SignalSource=SimulationProject 3637
EventTableTriggerIO 11577: Operator=0, IOValue=[1], IRC5Controller=? -1, SignalSource=SimulationProject 3637
EventTableTriggerIO 11578: Operator=0, IOValue=[0], IRC5Controller=? -1, SignalSource=SimulationProject 3637
EventTableTriggerIO 11579: Operator=0, IOValue=[0], IRC5Controller=? -1, SignalSource=SimulationProject 3637
EventTableTriggerIO 11580: Operator=0, IOValue=[1], IRC5Controller=? -1, SignalSource=SimulationProject 3637
EventTableTriggerIO 11581: Operator=0, IOValue=[1], IRC5Controller=? -1, SignalSource=SimulationProject 3637
EventTableTriggerIO 11582: Operator=0, IOValue=[0], IRC5Controller=? -1, SignalSource=SimulationProject 3637
EventTableTriggerIO 11583: Operator=0, IOValue=[0], IRC5Controller=? -1, SignalSource=SimulationProject 3637
EventTableTriggerIO 11584: Operator=0, IOValue=[1], IRC5Controller=? -1, SignalSource=SimulationProject 3637
EventTableTriggerIO 11585: Operator=0, IOValue=[1], IRC5Controller=? -1, SignalSource=SimulationProject 3637
EventTableTriggerIO 11586: Operator=0, IOValue=[0], IRC5Controller=? -1, SignalSource=SimulationProject 3637
EventTableTriggerIO 11587: Operator=0, IOValue=[0], IRC5Controller=? -1, SignalSource=SimulationProject 3637
EventTableTriggerIO 11588: Operator=0, IOValue=[1], IRC5Controller=? -1, SignalSource=SimulationProject 3637
EventTableTriggerIO 11589: Operator=0, IOValue=[1], IRC5Controller=? -1, SignalSource=SimulationProject 3637
EventTableTriggerIO 11590: Operator=0, IOValue=[0], IRC5Controller=? -1, SignalSource=SimulationProject 3637
EventTableTriggerIO 11591: Operator=0, IOValue=[0], IRC5Controller=? -1, SignalSource=SimulationProject 3637
EventTableTriggerIO 11592: Operator=0, IOValue=[1], IRC5Controller=? -1, SignalSource=SimulationProject 3637
EventTableTriggerIO 11593: Operator=0, IOValue=[1], IRC5Controller=? -1, SignalSource=SimulationProject 3637
EventTableTriggerIO 11594: Operator=0, IOValue=[0], IRC5Controller=? -1, SignalSource=SimulationProject 3637
EventTableTriggerIO 11595: Operator=0, IOValue=[0], IRC5Controller=? -1, SignalSource=SimulationProject 3637
EventTableTriggerIO 11596: Operator=0, IOValue=[1], IRC5Controller=? -1, SignalSource=SimulationProject 3637
EventTableTriggerIO 11597: Operator=0, IOValue=[1], IRC5Controller=? -1, SignalSource=SimulationProject 3637
EventTableTriggerIO 11598: Operator=0, IOValue=[0], IRC5Controller=? -1, SignalSource=SimulationProject 3637
EventTableTriggerIO 11599: Operator=0, IOValue=[0], IRC5Controller=? -1, SignalSource=SimulationProject 3637
EventTableTriggerIO 11600: Operator=0, IOValue=[1], IRC5Controller=? -1, SignalSource=SimulationProject 3637
EventTableTriggerIO 11601: Operator=0, IOValue=[1], IRC5Controller=? -1, SignalSource=SimulationProject 3637
EventTableTriggerIO 11602: Operator=0, IOValue=[0], IRC5Controller=? -1, SignalSource=SimulationProject 3637
EventTableTriggerIO 11603: Operator=0, IOValue=[0], IRC5Controller=? -1, SignalSource=SimulationProject 3637
EventTableTriggerIO 11604: Operator=0, IOValue=[1], IRC5Controller=? -1, SignalSource=SimulationProject 3637
EventTableTriggerIO 11605: Operator=0, IOValue=[1], IRC5Controller=? -1, SignalSource=SimulationProject 3637
EventTableTriggerIO 11606: Operator=0, IOValue=[0], IRC5Controller=? -1, SignalSource=SimulationProject 3637
EventTableTriggerIO 11607: Operator=0, IOValue=[0], IRC5Controller=? -1, SignalSource=SimulationProject 3637
EventTableTriggerIO 11608: Operator=0, IOValue=[1], IRC5Controller=? -1, SignalSource=SimulationProject 3637
EventTableTriggerIO 11609: Operator=0, IOValue=[1], IRC5Controller=? -1, SignalSource=SimulationProject 3637
EventTableTriggerIO 11610: Operator=0, IOValue=[0], IRC5Controller=? -1, SignalSource=SimulationProject 3637
EventTableTriggerIO 11611: Operator=0, IOValue=[0], IRC5Controller=? -1, SignalSource=SimulationProject 3637
EventTableTriggerIO 11612: Operator=0, IOValue=[1], IRC5Controller=? -1, SignalSource=SimulationProject 3637
EventTableTriggerIO 11613: Operator=0, IOValue=[1], IRC5Controller=? -1, SignalSource=SimulationProject 3637
EventTableTriggerIO 11614: Operator=0, IOValue=[0], IRC5Controller=? -1, SignalSource=SimulationProject 3637
EventTableTriggerIO 11615: Operator=0, IOValue=[0], IRC5Controller=? -1, SignalSource=SimulationProject 3637
EventTableTriggerIO 11616: Operator=0, IOValue=[1], IRC5Controller=? -1, SignalSource=SimulationProject 3637
EventTableTriggerIO 11617: Operator=0, IOValue=[1], IRC5Controller=? -1, SignalSource=SimulationProject 3637
EventTableTriggerIO 11618: Operator=0, IOValue=[0], IRC5Controller=? -1, SignalSource=SimulationProject 3637
EventTableTriggerIO 11619: Operator=0, IOValue=[0], IRC5Controller=? -1, SignalSource=SimulationProject 3637
EventTableTriggerIO 11620: Operator=0, IOValue=[1], IRC5Controller=? -1, SignalSource=SimulationProject 3637
EventTableTriggerIO 11621: Operator=0, IOValue=[1], IRC5Controller=? -1, SignalSource=SimulationProject 3637
EventTableTriggerIO 11622: Operator=0, IOValue=[0], IRC5Controller=? -1, SignalSource=SimulationProject 3637
EventTableTriggerIO 11623: Operator=0, IOValue=[0], IRC5Controller=? -1, SignalSource=SimulationProject 3637
EventTableTriggerIO 11624: Operator=0, IOValue=[1], IRC5Controller=? -1, SignalSource=SimulationProject 3637
EventTableTriggerIO 11625: Operator=0, IOValue=[1], IRC5Controller=? -1, SignalSource=SimulationProject 3637
EventTableTriggerIO 11626: Operator=0, IOValue=[0], IRC5Controller=? -1, SignalSource=SimulationProject 3637
EventTableTriggerIO 11627: Operator=0, IOValue=[0], IRC5Controller=? -1, SignalSource=SimulationProject 3637
EventTableTriggerIO 11628: Operator=0, IOValue=[1], IRC5Controller=? -1, SignalSource=SimulationProject 3637
EventTableTriggerIO 11629: Operator=0, IOValue=[1], IRC5Controller=? -1, SignalSource=SimulationProject 3637
EventTableTriggerIO 11630: Operator=0, IOValue=[0], IRC5Controller=? -1, SignalSource=SimulationProject 3637
EventTableTriggerIO 11631: Operator=0, IOValue=[0], IRC5Controller=? -1, SignalSource=SimulationProject 3637
EventTableTriggerIO 11632: Operator=0, IOValue=[1], IRC5Controller=? -1, SignalSource=SimulationProject 3637
EventTableTriggerIO 11633: Operator=0, IOValue=[1], IRC5Controller=? -1, SignalSource=SimulationProject 3637
EventTableTriggerIO 11634: Operator=0, IOValue=[0], IRC5Controller=? -1, SignalSource=SimulationProject 3637
EventTableTriggerIO 11635: Operator=0, IOValue=[0], IRC5Controller=? -1, SignalSource=SimulationProject 3637
EventTableTriggerIO 11636: Operator=0, IOValue=[1], IRC5Controller=? -1, SignalSource=SimulationProject 3637
EventTableTriggerIO 11637: Operator=0, IOValue=[1], IRC5Controller=? -1, SignalSource=SimulationProject 3637
EventTableTriggerIO 11638: Operator=0, IOValue=[0], IRC5Controller=? -1, SignalSource=SimulationProject 3637
EventTableTriggerIO 11639: Operator=0, IOValue=[0], IRC5Controller=? -1, SignalSource=SimulationProject 3637
EventTableEntry 11679: ActivationMode=2, Cyclic=false, Group=, Trigger=doStackTool_L 11680, Actions=[EventTableActionAttach 11681], Comment=
EventTableTriggerIO 11680: Operator=0, IOValue=[1], IRC5Controller=? -1, SignalSource=SimulationProject 3637
EventTableActionAttach 11681: MountObject=false, FlangeIndext=0, FindNearest=false, AttachmentParent=IRB6660_100_335__01_L 3595, AttachmentChild=StackTool 5990, Offset=[X=1, Y=0, Z=0, W=0, X=0, Y=1, Z=0, W=0, X=0, Y=0, Z=1, W=0, X=0, Y=0, Z=0, W=1]
EventTableEntry 11682: ActivationMode=2, Cyclic=false, Group=, Trigger=doStackTool_L 11683, Actions=[EventTableActionDetach 11684], Comment=
EventTableTriggerIO 11683: Operator=0, IOValue=[0], IRC5Controller=? -1, SignalSource=SimulationProject 3637
EventTableActionDetach 11684: AttachmentParent=IRB6660_100_335__01_L 3595, AttachmentChild=StackTool 5990
EventTableEntry 11685: ActivationMode=2, Cyclic=false, Group=, Trigger=doStack_L 11686, Actions=[EventTableActionAttach 11687], Comment=
EventTableTriggerIO 11686: Operator=0, IOValue=[1], IRC5Controller=? -1, SignalSource=SimulationProject 3637
EventTableActionAttach 11687: MountObject=false, FlangeIndext=0, FindNearest=true, AttachmentParent=StackTool 5990, AttachmentChild=? -1, Offset=[X=1, Y=0, Z=0, W=0, X=0, Y=1, Z=0, W=0, X=0, Y=0, Z=1, W=0, X=0, Y=0, Z=0, W=1]
EventTableEntry 11688: ActivationMode=2, Cyclic=false, Group=, Trigger=doStack_L 11689, Actions=[EventTableActionDetach 11690, EventTableActionAttach 12123], Comment=
EventTableTriggerIO 11689: Operator=0, IOValue=[0], IRC5Controller=? -1, SignalSource=SimulationProject 3637
EventTableActionDetach 11690: AttachmentParent=StackTool 5990, AttachmentChild=? -1
EventTableTriggerIO 11999: Operator=0, IOValue=[1], IRC5Controller=? -1, SignalSource=SimulationProject 3637
EventTableTriggerIO 12000: Operator=0, IOValue=[0], IRC5Controller=? -1, SignalSource=SimulationProject 3637
EventTableTriggerIO 12001: Operator=0, IOValue=[1], IRC5Controller=? -1, SignalSource=SimulationProject 3637
EventTableTriggerIO 12002: Operator=0, IOValue=[0], IRC5Controller=? -1, SignalSource=SimulationProject 3637
EventTableTriggerIO 12003: Operator=0, IOValue=[1], IRC5Controller=? -1, SignalSource=SimulationProject 3637
EventTableTriggerIO 12004: Operator=0, IOValue=[0], IRC5Controller=? -1, SignalSource=SimulationProject 3637
EventTableTriggerIO 12005: Operator=0, IOValue=[1], IRC5Controller=? -1, SignalSource=SimulationProject 3637
EventTableTriggerIO 12006: Operator=0, IOValue=[0], IRC5Controller=? -1, SignalSource=SimulationProject 3637
EventTableTriggerIO 12007: Operator=0, IOValue=[1], IRC5Controller=? -1, SignalSource=SimulationProject 3637
EventTableTriggerIO 12008: Operator=0, IOValue=[0], IRC5Controller=? -1, SignalSource=SimulationProject 3637
EventTableTriggerIO 12009: Operator=0, IOValue=[1], IRC5Controller=? -1, SignalSource=SimulationProject 3637
EventTableTriggerIO 12010: Operator=0, IOValue=[0], IRC5Controller=? -1, SignalSource=SimulationProject 3637
EventTableTriggerIO 12011: Operator=0, IOValue=[1], IRC5Controller=? -1, SignalSource=SimulationProject 3637
EventTableTriggerIO 12012: Operator=0, IOValue=[0], IRC5Controller=? -1, SignalSource=SimulationProject 3637
EventTableTriggerIO 12013: Operator=0, IOValue=[1], IRC5Controller=? -1, SignalSource=SimulationProject 3637
EventTableTriggerIO 12014: Operator=0, IOValue=[0], IRC5Controller=? -1, SignalSource=SimulationProject 3637
EventTableTriggerIO 12015: Operator=0, IOValue=[1], IRC5Controller=? -1, SignalSource=SimulationProject 3637
EventTableTriggerIO 12016: Operator=0, IOValue=[0], IRC5Controller=? -1, SignalSource=SimulationProject 3637
EventTableTriggerIO 12017: Operator=0, IOValue=[1], IRC5Controller=? -1, SignalSource=SimulationProject 3637
EventTableTriggerIO 12018: Operator=0, IOValue=[0], IRC5Controller=? -1, SignalSource=SimulationProject 3637
EventTableTriggerIO 12019: Operator=0, IOValue=[1], IRC5Controller=? -1, SignalSource=SimulationProject 3637
EventTableTriggerIO 12020: Operator=0, IOValue=[0], IRC5Controller=? -1, SignalSource=SimulationProject 3637
EventTableTriggerIO 12021: Operator=0, IOValue=[1], IRC5Controller=? -1, SignalSource=SimulationProject 3637
EventTableTriggerIO 12022: Operator=0, IOValue=[0], IRC5Controller=? -1, SignalSource=SimulationProject 3637
EventTableTriggerIO 12023: Operator=0, IOValue=[1], IRC5Controller=? -1, SignalSource=SimulationProject 3637
EventTableTriggerIO 12024: Operator=0, IOValue=[0], IRC5Controller=? -1, SignalSource=SimulationProject 3637
EventTableTriggerIO 12025: Operator=0, IOValue=[1], IRC5Controller=? -1, SignalSource=SimulationProject 3637
EventTableTriggerIO 12026: Operator=0, IOValue=[0], IRC5Controller=? -1, SignalSource=SimulationProject 3637
EventTableTriggerIO 12027: Operator=0, IOValue=[1], IRC5Controller=? -1, SignalSource=SimulationProject 3637
EventTableTriggerIO 12028: Operator=0, IOValue=[0], IRC5Controller=? -1, SignalSource=SimulationProject 3637
EventTableTriggerIO 12029: Operator=0, IOValue=[1], IRC5Controller=? -1, SignalSource=SimulationProject 3637
EventTableTriggerIO 12030: Operator=0, IOValue=[0], IRC5Controller=? -1, SignalSource=SimulationProject 3637
EventTableTriggerIO 12031: Operator=0, IOValue=[1], IRC5Controller=? -1, SignalSource=SimulationProject 3637
EventTableTriggerIO 12032: Operator=0, IOValue=[0], IRC5Controller=? -1, SignalSource=SimulationProject 3637
EventTableTriggerIO 12033: Operator=0, IOValue=[1], IRC5Controller=? -1, SignalSource=SimulationProject 3637
EventTableTriggerIO 12034: Operator=0, IOValue=[0], IRC5Controller=? -1, SignalSource=SimulationProject 3637
EventTableTriggerIO 12035: Operator=0, IOValue=[1], IRC5Controller=? -1, SignalSource=SimulationProject 3637
EventTableTriggerIO 12036: Operator=0, IOValue=[0], IRC5Controller=? -1, SignalSource=SimulationProject 3637
EventTableTriggerIO 12037: Operator=0, IOValue=[1], IRC5Controller=? -1, SignalSource=SimulationProject 3637
EventTableTriggerIO 12038: Operator=0, IOValue=[0], IRC5Controller=? -1, SignalSource=SimulationProject 3637
EventTableActionAttach 12123: MountObject=false, FlangeIndext=0, FindNearest=true, AttachmentParent=train_body 3634, AttachmentChild=? -1, Offset=[X=1, Y=0, Z=0, W=0, X=0, Y=1, Z=0, W=0, X=0, Y=0, Z=1, W=0, X=0, Y=0, Z=0, W=1]
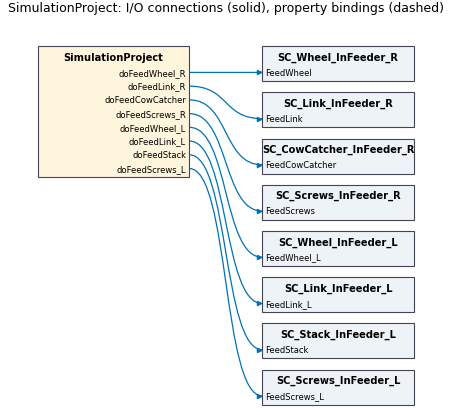
Station logic (signal -> signal, property => property):
  SimulationProject.doFeedWheel_R -> SC_Wheel_InFeeder_R.FeedWheel
  SimulationProject.doFeedLink_R -> SC_Link_InFeeder_R.FeedLink
  SimulationProject.doFeedCowCatcher -> SC_CowCatcher_InFeeder_R.FeedCowCatcher
  SimulationProject.doFeedScrews_R -> SC_Screws_InFeeder_R.FeedScrews
  SimulationProject.doFeedWheel_L -> SC_Wheel_InFeeder_L.FeedWheel_L
  SimulationProject.doFeedLink_L -> SC_Link_InFeeder_L.FeedLink_L
  SimulationProject.doFeedStack -> SC_Stack_InFeeder_L.FeedStack
  SimulationProject.doFeedScrews_L -> SC_Screws_InFeeder_L.FeedScrews_L

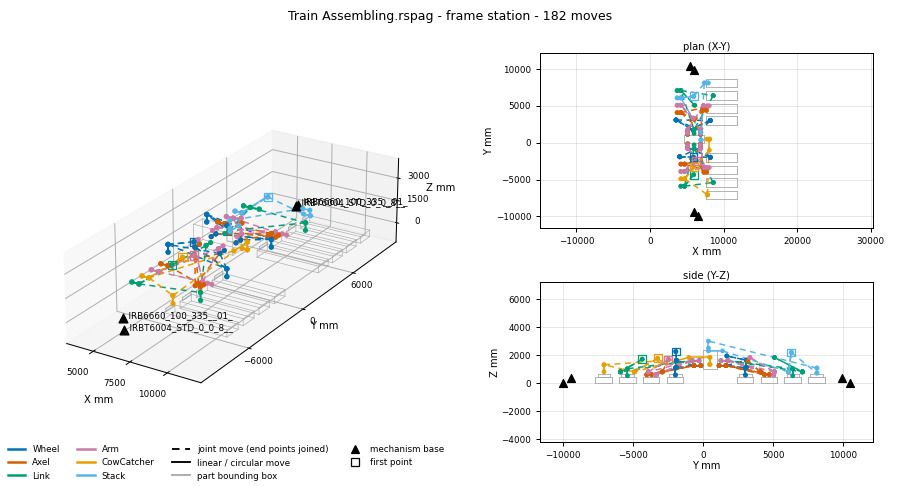
[picture p0: tool path of Train Assembling.rspag in frame station, 182 of 182 moves have a stored position in this frame; points joined in program order, loops and branches not executed]
--- Controller Data/SimulationProject/RAPID/TASK1/PROGMOD/CalibData.mod ---
MODULE CalibData
    PERS tooldata WheelTool:=[TRUE,[[0,0,380],[1,0,0,0]],[1,[0,0,1],[1,0,0,0],0,0,0]];
    PERS tooldata LinkTool:=[TRUE,[[0,-15.353,170],[1,0,0,0]],[1,[0,0,1],[1,0,0,0],0,0,0]];
    PERS tooldata CowCatcherTool:=[TRUE,[[-12.656,0,240],[1,0,0,0]],[1,[0,0,1],[1,0,0,0],0,0,0]];
    PERS tooldata AxelPinTool:=[TRUE,[[0,0,262.488],[1,0,0,0]],[1,[0,0,1],[1,0,0,0],0,0,0]];
    PERS tooldata ArmPinTool:=[TRUE,[[-1.688,0,169.608],[1,0,0,0]],[1,[0,0,1],[1,0,0,0],0,0,0]];
ENDMODULE

--- Controller Data/SimulationProject/RAPID/TASK1/PROGMOD/MainModule.mod ---
MODULE MainModule
    TASK PERS wobjdata Workobject_R:=[FALSE,TRUE,"",[[9409.5,1350,665.5],[0.5,0.5,-0.5,-0.5]],[[0,0,0],[1,0,0,0]]];
ENDMODULE

--- Controller Data/SimulationProject/RAPID/TASK1/PROGMOD/Module1.mod ---
MODULE Module1
    CONST robtarget pWheel_Home:=[[1242.824180666,1202.379933267,1943.391267721],[0.252183059,0.41980817,-0.758652436,0.429664156],[0,-3,2,0],[5000,9E+09,9E+09,9E+09,9E+09,9E+09]];
    CONST robtarget pWheelTool_App:=[[-625,580,1900],[0.707106781,0.707106781,0,0],[0,0,-1,0],[6000,9E+09,9E+09,9E+09,9E+09,9E+09]];
    CONST robtarget pWheelTool:=[[-625,80,1900],[0.707106781,0.707106781,0,0],[0,0,-1,0],[6000,9E+09,9E+09,9E+09,9E+09,9E+09]];
    CONST robtarget pWheelPick_App:=[[3526.022,27.115,1968.551],[0,0,-0.707106781,0.707106781],[-1,0,0,0],[6000,9E+09,9E+09,9E+09,9E+09,9E+09]];
    CONST robtarget pWheelPick:=[[3526.022,-472.885,1968.551],[0,0,-0.707106781,0.707106781],[-1,0,0,0],[6000,9E+09,9E+09,9E+09,9E+09,9E+09]];
    CONST robtarget pWheelPlace_App:=[[450,200,650],[0,-0.707106781,0.707106781,0],[0,0,-1,0],[6000,9E+09,9E+09,9E+09,9E+09,9E+09]];
    CONST robtarget pWheelPlace:=[[450,200,150],[0,-0.707106781,0.707106781,0],[0,0,-1,0],[6000,9E+09,9E+09,9E+09,9E+09,9E+09]];
    CONST robtarget pWheelPlace2:=[[2200,200,150],[0,-0.707106781,0.707106781,0],[-1,1,-2,0],[6000,9E+09,9E+09,9E+09,9E+09,9E+09]];
    CONST robtarget pWheelPlace2_App:=[[2200,200,650],[0,-0.707106781,0.707106781,0],[-1,1,-2,0],[6000,9E+09,9E+09,9E+09,9E+09,9E+09]];
    CONST robtarget pWheelPlace1_App:=[[450,200,650],[0,-0.707106781,0.707106781,0],[0,0,-1,0],[6000,9E+09,9E+09,9E+09,9E+09,9E+09]];
    CONST robtarget pWheelPlace1:=[[450,200,150],[0,-0.707106781,0.707106781,0],[0,0,-1,0],[6000,9E+09,9E+09,9E+09,9E+09,9E+09]];
    CONST robtarget pAxelTool_App:=[[25,-250,2900],[0.707106781,0.707106781,0,0],[0,0,-1,0],[5000,9E+09,9E+09,9E+09,9E+09,9E+09]];
    CONST robtarget pAxelTool:=[[-475,-250,2900],[0.707106781,0.707106781,0,0],[0,0,-1,0],[5000,9E+09,9E+09,9E+09,9E+09,9E+09]];
    CONST robtarget pAxelPick1_App:=[[2662.532,-450.037,3664.742],[0.5,-0.5,0.5,-0.5],[-1,0,-1,0],[4500,9E+09,9E+09,9E+09,9E+09,9E+09]];
    CONST robtarget pAxelPick1:=[[3012.532,-450.037,3664.742],[0.5,-0.5,0.5,-0.5],[-1,0,-1,0],[4500,9E+09,9E+09,9E+09,9E+09,9E+09]];
    CONST robtarget pAxelPlace1_App:=[[450,200,650],[0,-0.707106781,0.707106781,0],[0,0,-1,0],[6000,9E+09,9E+09,9E+09,9E+09,9E+09]];
    CONST robtarget pAxelPlace1:=[[450,200,150],[0,-0.707106781,0.707106781,0],[0,0,-1,0],[6000,9E+09,9E+09,9E+09,9E+09,9E+09]];
    CONST robtarget pAxelPick2_App:=[[2662.532,-450.037,4014.742],[0.5,-0.5,0.5,-0.5],[-1,0,-1,0],[4500,9E+09,9E+09,9E+09,9E+09,9E+09]];
    CONST robtarget pAxelPick2:=[[3012.532,-450.037,4014.742],[0.5,-0.5,0.5,-0.5],[-1,0,-1,0],[4500,9E+09,9E+09,9E+09,9E+09,9E+09]];
    CONST robtarget pAxelPlace2_App:=[[2200,199.999,650],[0,-0.707106781,0.707106781,0],[-1,-1,0,0],[6000,9E+09,9E+09,9E+09,9E+09,9E+09]];
    CONST robtarget pAxelPlace2:=[[2200,199.999,150],[0,-0.707106781,0.707106781,0],[-1,-1,0,0],[6000,9E+09,9E+09,9E+09,9E+09,9E+09]];
    CONST robtarget pAxel_Home:=[[1589.533728527,623.070993853,2474.769248489],[0.078664167,-0.743773001,0.663630968,0.01440867],[-1,-1,-1,0],[4500,9E+09,9E+09,9E+09,9E+09,9E+09]];
    CONST robtarget pLink_Home:=[[1265.765540179,653.585946858,4340.972053129],[0.621057404,0.765826467,-0.132334037,0.101416105],[0,0,-1,0],[3000,9E+09,9E+09,9E+09,9E+09,9E+09]];
    CONST robtarget pLinkTool_App:=[[25,-250,5900],[0.707106781,0.707106781,0,0],[0,0,-1,0],[3000,9E+09,9E+09,9E+09,9E+09,9E+09]];
    CONST robtarget pLinkTool:=[[-475,-250,5900],[0.707106781,0.707106781,0,0],[0,0,-1,0],[3000,9E+09,9E+09,9E+09,9E+09,9E+09]];
    CONST robtarget pLinkPick_App:=[[3923.322,-28.104,5395.576],[0.5,0.5,-0.5,0.5],[-1,0,-1,0],[3000,9E+09,9E+09,9E+09,9E+09,9E+09]];
    CONST robtarget pLinkPick:=[[3923.322,-528.104,5395.576],[0.5,0.5,-0.5,0.5],[-1,0,-1,0],[3000,9E+09,9E+09,9E+09,9E+09,9E+09]];
    CONST robtarget pLinkPlace_App:=[[1325,549.999,774.937],[0,-0.707106781,0.707106781,0],[0,0,-1,0],[6000,9E+09,9E+09,9E+09,9E+09,9E+09]];
    CONST robtarget pLinkPlace:=[[1325,549.999,274.937],[0,-0.707106781,0.707106781,0],[0,0,-1,0],[6000,9E+09,9E+09,9E+09,9E+09,9E+09]];
    CONST robtarget pArm_Home:=[[1589.533728527,623.070993853,2474.769248489],[0.078664167,-0.743773001,0.663630968,0.01440867],[-1,1,-3,0],[4500,9E+09,9E+09,9E+09,9E+09,9E+09]];
    CONST robtarget pArmTool_App:=[[23.312,-251.508,3900],[0.707106781,0.707106781,0,0],[0,2,-3,0],[4500,9E+09,9E+09,9E+09,9E+09,9E+09]];
    CONST robtarget pArmTool:=[[-476.688,-251.508,3900],[0.707106781,0.707106781,0,0],[0,2,-3,0],[4500,9E+09,9E+09,9E+09,9E+09,9E+09]];
    CONST robtarget pArmPick_App:=[[2757.032,-450.037,3364.742],[0.5,-0.5,0.5,-0.5],[-1,0,-1,0],[4500,9E+09,9E+09,9E+09,9E+09,9E+09]];
    CONST robtarget pArmPick1:=[[3087.032,-450.037,3364.742],[0.5,-0.5,0.5,-0.5],[-1,0,-1,0],[4500,9E+09,9E+09,9E+09,9E+09,9E+09]];
    CONST robtarget pArmPlace1_App:=[[450,549.999,789.937],[0,-0.707106781,0.707106781,0],[0,0,-1,0],[6000,9E+09,9E+09,9E+09,9E+09,9E+09]];
    CONST robtarget pArmPlace1:=[[450,549.999,289.937],[0,-0.707106781,0.707106781,0],[0,0,-1,0],[6000,9E+09,9E+09,9E+09,9E+09,9E+09]];
    CONST robtarget pArmPick2:=[[3387.032,-450.037,3364.742],[0.5,-0.5,0.5,-0.5],[-1,0,-1,0],[4500,9E+09,9E+09,9E+09,9E+09,9E+09]];
    CONST robtarget pArmPlace2_App:=[[2200,549.999,790],[0,-0.707106781,0.707106781,0],[-1,1,-2,0],[6000,9E+09,9E+09,9E+09,9E+09,9E+09]];
    CONST robtarget pArmPlace2:=[[2200,549.999,290],[0,-0.707106781,0.707106781,0],[-1,1,-2,0],[6000,9E+09,9E+09,9E+09,9E+09,9E+09]];
    CONST robtarget pCow_Home:=[[1277.263853357,716.038961172,3233.744403976],[0.300792033,0.623356768,0.641631509,-0.330544246],[0,0,1,0],[4500,9E+09,9E+09,9E+09,9E+09,9E+09]];
    CONST robtarget pCowTool_App:=[[45,-250,4900],[0,0,-0.707106781,0.707106781],[0,0,1,0],[4500,9E+09,9E+09,9E+09,9E+09,9E+09]];
    CONST robtarget pCowTool:=[[-455,-250,4900],[0,0,-0.707106781,0.707106781],[0,0,1,0],[4500,9E+09,9E+09,9E+09,9E+09,9E+09]];
    CONST robtarget pCowPick_App:=[[3147.835,256.362,7068.449],[0.707106781,0.707106781,0,0],[-1,0,-2,0],[2000,9E+09,9E+09,9E+09,9E+09,9E+09]];
    CONST robtarget pCowPick:=[[3147.835,-243.638,7068.449],[0.707106781,0.707106781,0,0],[-1,0,-2,0],[2000,9E+09,9E+09,9E+09,9E+09,9E+09]];
    CONST robtarget pCowPlace_App:=[[3405,782.5,-490],[0,0,-0.707106781,0.707106781],[-1,0,-4,0],[7600,9E+09,9E+09,9E+09,9E+09,9E+09]];
    CONST robtarget pCowPlace:=[[3055,282.5,-490],[0,0,-0.707106781,0.707106781],[-1,0,-4,0],[7600,9E+09,9E+09,9E+09,9E+09,9E+09]];
    CONST robtarget pCowPlace_App2:=[[3405,282.5,-490],[0,0,-0.707106781,0.707106781],[-1,0,-4,0],[7600,9E+09,9E+09,9E+09,9E+09,9E+09]];
    CONST robtarget pCowPlace_App3:=[[3405,782.5,1010],[0,0,-0.707106781,0.707106781],[-1,0,-4,0],[7600,9E+09,9E+09,9E+09,9E+09,9E+09]];
    !***********************************************************
    !
    ! Module:  Module1
    !
    ! Description:
    !   <Insert description here>
    !
    ! Author: DELL
    !
    ! Version: 1.0
    !
    !***********************************************************


    !***********************************************************
    !
    ! Procedure main
    !
    !   This is the entry point of your program
    !
    !***********************************************************
    PROC main()
        Reset doFeedWheel_R;
        Reset doFeedLink_R;
        Reset doFeedScrews_R;
        Reset doFeedCowCatcher;
        Reset doWheelTool;
        Reset doWheel;
        Reset doAxel;
        Reset doAxelTool;
        Reset doLinkTool;
        Reset doLink;
        Reset doArmTool;
        Reset doArm;
        Reset doCowTool;
        Reset doCow;

        SetDO doFeedWheel_R,1;
        SetDO doFeedLink_R,1;
        SetDO doFeedScrews_R,1;
        SetDO doFeedCowCatcher,1;

        WHILE TRUE DO
            Reset doFeedWheel_R;
            Reset doFeedLink_R;
            Reset doFeedScrews_R;
            Reset doFeedCowCatcher;
            Reset doWheelTool;
            Reset doWheel;
            Reset doAxel;
            Reset doAxelTool;
            Reset doLinkTool;
            Reset doLink;
            Reset doArmTool;
            Reset doArm;
            Reset doCowTool;
            Reset doCow;

            Wheel;
            Axel;
            Link;
            Arm;
            CowCatcher;
        ENDWHILE
    ENDPROC

    PROC Wheel()
        MoveJ pWheel_Home,v1000,z100,tool0\WObj:=Workobject_R;
        MoveJ pWheelTool_App,v1000,fine,tool0\WObj:=Workobject_R;
        MoveL pWheelTool,v500,fine,tool0\WObj:=Workobject_R;
        SetDO doWheelTool,1;
        WaitTime 1;
        MoveL pWheelTool_App,v500,fine,WheelTool\WObj:=Workobject_R;
        MoveJ pWheelPick_App,v1000,fine,WheelTool\WObj:=Workobject_R;
        MoveL pWheelPick,v500,fine,WheelTool\WObj:=Workobject_R;
        SetDO doWheel,1;
        Reset doFeedWheel_R;
        SetDO doFeedWheel_R,1;
        WaitTime 1;
        MoveL pWheelPick_App,v500,fine,WheelTool\WObj:=Workobject_R;
        MoveJ pWheelPlace1_App,v1000,fine,WheelTool\WObj:=Workobject_R;
        MoveL pWheelPlace1,v200,fine,WheelTool\WObj:=Workobject_R;
        SetDO doWheel,0;
        WaitTime 1;
        MoveL pWheelPlace1_App,v200,fine,WheelTool\WObj:=Workobject_R;
        MoveJ pWheelPick_App,v1000,fine,WheelTool\WObj:=Workobject_R;
        MoveL pWheelPick,v500,fine,WheelTool\WObj:=Workobject_R;
        SetDO doWheel,1;
        Reset doFeedWheel_R;
        SetDO doFeedWheel_R,1;
        WaitTime 1;
        MoveL pWheelPick_App,v500,fine,WheelTool\WObj:=Workobject_R;
        MoveJ pWheelPlace2_App,v1000,fine,WheelTool\WObj:=Workobject_R;
        MoveL pWheelPlace2,v200,fine,WheelTool\WObj:=Workobject_R;
        SetDO doWheel,0;
        WaitTime 1;
        MoveL pWheelPlace2_App,v200,fine,WheelTool\WObj:=Workobject_R;
        MoveJ pWheelTool_App,v1000,fine,WheelTool\WObj:=Workobject_R;
        MoveL pWheelTool,v1000,fine,tool0\WObj:=Workobject_R;
        SetDO doWheelTool,0;
        WaitTime 1;
        MoveL pWheelTool_App,v1000,fine,tool0\WObj:=Workobject_R;
        MoveJ pWheel_Home,v1000,z100,tool0\WObj:=Workobject_R;
    ENDPROC

    PROC Axel()
        MoveJ pAxel_Home,v1000,z100,tool0\WObj:=Workobject_R;
        MoveJ pAxelTool_App,v1000,fine,tool0\WObj:=Workobject_R;
        MoveL pAxelTool,v500,fine,tool0\WObj:=Workobject_R;
        SetDO doAxelTool,1;
        WaitTime 1;
        MoveL pAxelTool_App,v500,fine,tool0\WObj:=Workobject_R;
        MoveJ pAxelPick1_App,v1000,fine,AxelPinTool\WObj:=Workobject_R;
        MoveL pAxelPick1,v500,fine,AxelPinTool\WObj:=Workobject_R;
        SetDO doAxel,1;
        WaitTime 1;
        MoveL pAxelPick1_App,v500,fine,AxelPinTool\WObj:=Workobject_R;
        MoveJ pAxelPlace1_App,v1000,fine,AxelPinTool\WObj:=Workobject_R;
        MoveL pAxelPlace1,v200,fine,AxelPinTool\WObj:=Workobject_R;
        SetDO doAxel,0;
        WaitTime 1;
        MoveL pAxelPlace1_App,v200,fine,AxelPinTool\WObj:=Workobject_R;
        MoveJ pAxelPick2_App,v1000,fine,AxelPinTool\WObj:=Workobject_R;
        MoveL pAxelPick2,v500,fine,AxelPinTool\WObj:=Workobject_R;
        SetDO doAxel,1;
        WaitTime 1;
        MoveL pAxelPick2_App,v500,fine,AxelPinTool\WObj:=Workobject_R;
        MoveJ pAxelPlace2_App,v1000,fine,AxelPinTool\WObj:=Workobject_R;
        MoveL pAxelPlace2,v200,fine,AxelPinTool\WObj:=Workobject_R;
        SetDO doAxel,0;
        WaitTime 1;
        MoveL pAxelPlace2_App,v200,fine,AxelPinTool\WObj:=Workobject_R;
        MoveJ pAxelTool_App,v1000,fine,tool0\WObj:=Workobject_R;
        MoveL pAxelTool,v500,fine,tool0\WObj:=Workobject_R;
        SetDO doAxelTool,0;
        WaitTime 1;
        MoveL pAxelTool_App,v500,fine,tool0\WObj:=Workobject_R;
        MoveJ pAxel_Home,v1000,z100,tool0\WObj:=Workobject_R;
    ENDPROC

    PROC Link()
        MoveJ pLink_Home,v1000,z100,tool0\WObj:=Workobject_R;
        MoveJ pLinkTool_App,v1000,fine,tool0\WObj:=Workobject_R;
        MoveL pLinkTool,v500,fine,tool0\WObj:=Workobject_R;
        SetDO doLinkTool,1;
        WaitTime 1;
        MoveL pLinkTool_App,v500,fine,tool0\WObj:=Workobject_R;
        MoveJ pLinkPick_App,v1000,fine,LinkTool\WObj:=Workobject_R;
        MoveL pLinkPick,v500,fine,LinkTool\WObj:=Workobject_R;
        SetDO doLink,1;
        WaitTime 1;
        MoveL pLinkPick_App,v500,fine,LinkTool\WObj:=Workobject_R;
        MoveJ pLinkPlace_App,v1000,z100,LinkTool\WObj:=Workobject_R;
        MoveL pLinkPlace,v200,fine,LinkTool\WObj:=Workobject_R;
        SetDO doLink,0;
        Reset doFeedLink_R;
        SetDO doFeedLink_R,1;
        WaitTime 1;
        MoveL pLinkPlace_App,v200,fine,LinkTool\WObj:=Workobject_R;
        MoveJ pLinkTool_App,v1000,fine,tool0\WObj:=Workobject_R;
        MoveL pLinkTool,v500,fine,tool0\WObj:=Workobject_R;
        SetDO doLinkTool,0;
        WaitTime 1;
        MoveL pLinkTool_App,v500,fine,tool0\WObj:=Workobject_R;
        MoveJ pLink_Home,v1000,z100,tool0\WObj:=Workobject_R;
    ENDPROC

    PROC Arm()
        MoveJ pArm_Home,v1000,z100,tool0\WObj:=Workobject_R;
        MoveJ pArmTool_App,v1000,fine,tool0\WObj:=Workobject_R;
        MoveL pArmTool,v500,fine,tool0\WObj:=Workobject_R;
        SetDO doArmTool,1;
        WaitTime 1;
        MoveL pArmTool_App,v500,fine,tool0\WObj:=Workobject_R;
        MoveJ pArmPick_App,v1000,fine,ArmPinTool\WObj:=Workobject_R;
        MoveL pArmPick1,v500,fine,ArmPinTool\WObj:=Workobject_R;
        SetDO doArm,1;
        WaitTime 1;
        MoveL pArmPick_App,v500,fine,ArmPinTool\WObj:=Workobject_R;
        MoveJ pArmPlace1_App,v1000,fine,ArmPinTool\WObj:=Workobject_R;
        MoveL pArmPlace1,v200,fine,ArmPinTool\WObj:=Workobject_R;
        SetDO doArm,0;
        WaitTime 1;
        MoveL pArmPlace1_App,v200,fine,ArmPinTool\WObj:=Workobject_R;
        MoveJ pArmPick_App,v1000,fine,ArmPinTool\WObj:=Workobject_R;
        MoveL pArmPick2,v500,fine,ArmPinTool\WObj:=Workobject_R;
        SetDO doArm,1;
        WaitTime 1;
        MoveL pArmPick_App,v500,fine,ArmPinTool\WObj:=Workobject_R;
        MoveJ pArmPlace2_App,v1000,fine,ArmPinTool\WObj:=Workobject_R;
        MoveL pArmPlace2,v500,fine,ArmPinTool\WObj:=Workobject_R;
        SetDO doArm,0;
        Reset doFeedScrews_R;
        SetDO doFeedScrews_R,1;
        WaitTime 1;
        MoveL pArmPlace2_App,v500,fine,ArmPinTool\WObj:=Workobject_R;
        MoveJ pArmTool_App,v1000,fine,tool0\WObj:=Workobject_R;
        MoveL pArmTool,v500,fine,tool0\WObj:=Workobject_R;
        SetDO doArmTool,0;
        WaitTime 1;
        MoveL pArmTool_App,v500,fine,tool0\WObj:=Workobject_R;
        MoveJ pArm_Home,v1000,z100,tool0\WObj:=Workobject_R;
    ENDPROC

    PROC CowCatcher()
        MoveJ pCow_Home,v1000,z100,tool0\WObj:=Workobject_R;
        MoveJ pCowTool_App,v1000,fine,tool0\WObj:=Workobject_R;
        MoveL pCowTool,v500,fine,tool0\WObj:=Workobject_R;
        SetDO doCowTool,1;
        WaitTime 1;
        MoveL pCowTool_App,v500,fine,tool0\WObj:=Workobject_R;
        MoveJ pCowPick_App,v1000,fine,CowCatcherTool\WObj:=Workobject_R;
        MoveL pCowPick,v500,fine,CowCatcherTool\WObj:=Workobject_R;
        SetDO doCow,1;
        Reset doFeedCowCatcher;
        SetDO doFeedCowCatcher,1;
        WaitTime 1;
        MoveL pCowPick_App,v500,fine,CowCatcherTool\WObj:=Workobject_R;
        MoveJ pCowPlace_App,v1000,fine,CowCatcherTool\WObj:=Workobject_R;
        MoveL pCowPlace_App2,v200,fine,CowCatcherTool\WObj:=Workobject_R;
        MoveL pCowPlace,v200,fine,CowCatcherTool\WObj:=Workobject_R;
        SetDO doCow,0;
        WaitTime 1;
        MoveL pCowPlace_App2,v500,fine,CowCatcherTool\WObj:=Workobject_R;
        MoveL pCowPlace_App,v200,fine,CowCatcherTool\WObj:=Workobject_R;
        MoveL pCowPlace_App3,v500,fine,CowCatcherTool\WObj:=Workobject_R;
        MoveJ pCowTool_App,v1000,fine,tool0\WObj:=Workobject_R;
        MoveL pCowTool,v500,fine,tool0\WObj:=Workobject_R;
        SetDO doCowTool,0;
        WaitTime 1;
        MoveL pCowTool_App,v500,fine,tool0\WObj:=Workobject_R;
        MoveJ pCow_Home,v1000,z100,tool0\WObj:=Workobject_R;
    ENDPROC
ENDMODULE

--- Controller Data/SimulationProject/RAPID/TASK2/PROGMOD/CalibData.mod ---
MODULE CalibData
    PERS tooldata ArmPinTool:=[TRUE,[[-1.688,0,169.608],[1,0,0,0]],[1,[0,0,1],[1,0,0,0],0,0,0]];
    PERS tooldata AxelPinTool:=[TRUE,[[0,0,262.488],[1,0,0,0]],[1,[0,0,1],[1,0,0,0],0,0,0]];
    PERS tooldata LinkTool:=[TRUE,[[0,-15.353,170],[1,0,0,0]],[1,[0,0,1],[1,0,0,0],0,0,0]];
    PERS tooldata StackTool:=[TRUE,[[0,0,634.007],[1,0,0,0]],[1,[0,0,1],[1,0,0,0],0,0,0]];
    PERS tooldata WheelTool:=[TRUE,[[0,0,380],[1,0,0,0]],[1,[0,0,1],[1,0,0,0],0,0,0]];
ENDMODULE

--- Controller Data/SimulationProject/RAPID/TASK2/PROGMOD/MainModule.mod ---
MODULE MainModule
    TASK PERS wobjdata Workobject_L:=[FALSE,TRUE,"",[[10409.5,1350,665.5],[0.5,0.5,-0.5,-0.5]],[[0,0,0],[1,0,0,0]]];
ENDMODULE

--- Controller Data/SimulationProject/RAPID/TASK2/PROGMOD/Module1.mod ---
MODULE Module1
    CONST robtarget pWheel_Home:=[[1210.604982417,886.176680686,-700.213209156],[0.808874476,-0.007470781,-0.02519747,-0.587393699],[-1,-1,0,0],[5300,9E+09,9E+09,9E+09,9E+09,9E+09]];
    CONST robtarget pWheelPick:=[[3526.022,-472.885,-2031.449],[0,0,-0.707106781,0.707106781],[0,0,-1,0],[5300,9E+09,9E+09,9E+09,9E+09,9E+09]];
    CONST robtarget pWheelPick_App:=[[3526.022,27.115,-2031.449],[0,0,-0.707106781,0.707106781],[0,0,-1,0],[5300,9E+09,9E+09,9E+09,9E+09,9E+09]];
    CONST robtarget pWheelPlace1_App:=[[450,200,-650],[0.707106781,0,0,-0.707106781],[-1,1,-2,0],[5300,9E+09,9E+09,9E+09,9E+09,9E+09]];
    CONST robtarget pWheelPlace1:=[[450,200,-150],[0.707106781,0,0,-0.707106781],[-1,1,-2,0],[5300,9E+09,9E+09,9E+09,9E+09,9E+09]];
    CONST robtarget pWheelPlace2:=[[2200,200,-150],[0.707106781,0,0,-0.707106781],[0,0,-1,0],[5300,9E+09,9E+09,9E+09,9E+09,9E+09]];
    CONST robtarget pWheelPlace2_App:=[[2200,200,-650],[0.707106781,0,0,-0.707106781],[0,0,-1,0],[5300,9E+09,9E+09,9E+09,9E+09,9E+09]];
    CONST robtarget pWheelTool:=[[-1125,80,-2100],[0.707106781,0.707106781,0,0],[-1,0,0,0],[5300,9E+09,9E+09,9E+09,9E+09,9E+09]];
    CONST robtarget pWheelTool_App:=[[-1125,580,-2100],[0.707106781,0.707106781,0,0],[-1,0,0,0],[5300,9E+09,9E+09,9E+09,9E+09,9E+09]];
    CONST robtarget pAxel_Home:=[[1331.946587742,530.401688848,-2202.999678157],[0.692258559,0.513979341,0.303902761,-0.405273286],[0,0,0,0],[4500,9E+09,9E+09,9E+09,9E+09,9E+09]];
    CONST robtarget pAxelPick1:=[[3012.532,-450.037,-3735.258],[0.5,-0.5,0.5,-0.5],[0,-1,0,0],[4200,9E+09,9E+09,9E+09,9E+09,9E+09]];
    CONST robtarget pAxelPick1_App:=[[2512.032,-450.037,-3735.258],[0.5,-0.5,0.5,-0.5],[0,-1,0,0],[4200,9E+09,9E+09,9E+09,9E+09,9E+09]];
    CONST robtarget pAxelPick2:=[[3012.532,-450.037,-3385.258],[0.5,-0.5,0.5,-0.5],[0,-1,0,0],[4500,9E+09,9E+09,9E+09,9E+09,9E+09]];
    CONST robtarget pAxelPick2_App:=[[2512.032,-450.037,-3385.258],[0.5,-0.5,0.5,-0.5],[0,-1,0,0],[4500,9E+09,9E+09,9E+09,9E+09,9E+09]];
    CONST robtarget pAxelPlace1:=[[450,199.999,-150],[0.707106781,0,0,-0.707106781],[-1,-1,0,0],[5300,9E+09,9E+09,9E+09,9E+09,9E+09]];
    CONST robtarget pAxelPlace1_App:=[[450,199.999,-650],[0.707106781,0,0,-0.707106781],[-1,-1,0,0],[5300,9E+09,9E+09,9E+09,9E+09,9E+09]];
    CONST robtarget pAxelPlace2:=[[2200,199.999,-150],[0.707106781,0,0,-0.707106781],[0,0,-1,0],[5300,9E+09,9E+09,9E+09,9E+09,9E+09]];
    CONST robtarget pAxelPlace2_App:=[[2200,199.999,-650],[0.707106781,0,0,-0.707106781],[0,0,-1,0],[5300,9E+09,9E+09,9E+09,9E+09,9E+09]];
    CONST robtarget pAxelTool:=[[-975,-250,-3100],[0.707106781,0.707106781,0,0],[-1,0,0,0],[4500,9E+09,9E+09,9E+09,9E+09,9E+09]];
    CONST robtarget pAxelTool_App:=[[-475,-250,-3100],[0.707106781,0.707106781,0,0],[-1,0,0,0],[4500,9E+09,9E+09,9E+09,9E+09,9E+09]];
    CONST robtarget pLink_Home:=[[1394.810040234,777.860574146,-4102.059903428],[0.776971008,0.59637092,0.127234498,-0.156426217],[0,0,0,0],[2500,9E+09,9E+09,9E+09,9E+09,9E+09]];
    CONST robtarget pLinkPick:=[[3923.322,-528.104,-5404.424],[0.5,0.5,0.5,-0.5],[0,0,0,0],[2500,9E+09,9E+09,9E+09,9E+09,9E+09]];
    CONST robtarget pLinkPick_App:=[[3923.322,-28.104,-5404.424],[0.5,0.5,0.5,-0.5],[0,0,0,0],[2500,9E+09,9E+09,9E+09,9E+09,9E+09]];
    CONST robtarget pLinkPlace:=[[1325,549.999,-275],[0.707106781,0,0,-0.707106781],[0,0,-1,0],[5500,9E+09,9E+09,9E+09,9E+09,9E+09]];
    CONST robtarget pLinkPlace_App:=[[1325,549.999,-775],[0.707106781,0,0,-0.707106781],[0,0,-1,0],[5500,9E+09,9E+09,9E+09,9E+09,9E+09]];
    CONST robtarget pLinkTool:=[[-975,-250,-6100],[0.707106781,0.707106781,0,0],[-1,0,0,0],[2500,9E+09,9E+09,9E+09,9E+09,9E+09]];
    CONST robtarget pLinkTool_App:=[[-475,-250,-6100],[0.707106781,0.707106781,0,0],[-1,0,0,0],[2500,9E+09,9E+09,9E+09,9E+09,9E+09]];
    CONST robtarget pArm_Home:=[[1195.214292362,772.250595684,-2352.468426474],[0.746978165,0.107136403,0.061630521,-0.653258824],[-1,0,0,0],[4200,9E+09,9E+09,9E+09,9E+09,9E+09]];
    CONST robtarget pArmPick1:=[[3092.032,-450.037,-4035.258],[0.5,-0.5,0.5,-0.5],[0,1,-2,0],[4200,9E+09,9E+09,9E+09,9E+09,9E+09]];
    CONST robtarget pArmPick2:=[[3392.032,-450.037,-4035.258],[0.5,-0.5,0.5,-0.5],[0,1,-2,0],[4200,9E+09,9E+09,9E+09,9E+09,9E+09]];
    CONST robtarget pArmPick_App:=[[2592.032,-450.037,-4035.258],[0.5,-0.5,0.5,-0.5],[0,1,-2,0],[4200,9E+09,9E+09,9E+09,9E+09,9E+09]];
    CONST robtarget pArmPlace1:=[[450,549.999,-284.978],[0.707106781,0,0,-0.707106781],[-1,1,-2,0],[5500,9E+09,9E+09,9E+09,9E+09,9E+09]];
    CONST robtarget pArmPlace1_App:=[[450,549.999,-784.978],[0.707106781,0,0,-0.707106781],[-1,1,-2,0],[5500,9E+09,9E+09,9E+09,9E+09,9E+09]];
    CONST robtarget pArmPlace2:=[[2200,549.999,-285],[0.707106781,0,0,-0.707106781],[0,2,-3,0],[5500,9E+09,9E+09,9E+09,9E+09,9E+09]];
    CONST robtarget pArmPlace2_App:=[[2200,549.999,-785],[0.707106781,0,0,-0.707106781],[0,2,-3,0],[5500,9E+09,9E+09,9E+09,9E+09,9E+09]];
    CONST robtarget pArmTool:=[[-976.688,-251.508,-4100],[0.707106781,0.707106781,0,0],[-1,0,0,0],[4200,9E+09,9E+09,9E+09,9E+09,9E+09]];
    CONST robtarget pArmTool_App:=[[-476.688,-251.508,-4100],[0.707106781,0.707106781,0,0],[-1,0,0,0],[4200,9E+09,9E+09,9E+09,9E+09,9E+09]];
    CONST robtarget pStack_Home:=[[1271.729574606,1132.366623981,-5305.875574751],[0.745766844,0.007420539,0.010320689,-0.666085755],[-1,-1,0,0],[500,9E+09,9E+09,9E+09,9E+09,9E+09]];
    CONST robtarget pStackTool_App:=[[-475,-250,-5100],[0.707106781,0.707106781,0,0],[-1,0,0,0],[3000,9E+09,9E+09,9E+09,9E+09,9E+09]];
    CONST robtarget pStackTool:=[[-975,-250,-5100],[0.707106781,0.707106781,0,0],[-1,0,0,0],[3000,9E+09,9E+09,9E+09,9E+09,9E+09]];
    CONST robtarget pStackPick1_App:=[[2769.153,-334.791,-7133.923],[0.5,-0.5,0.5,-0.5],[0,1,-2,0],[500,9E+09,9E+09,9E+09,9E+09,9E+09]];
    CONST robtarget pStackPick1:=[[3269.153,-334.791,-7133.923],[0.5,-0.5,0.5,-0.5],[0,1,-2,0],[500,9E+09,9E+09,9E+09,9E+09,9E+09]];
    CONST robtarget pStackPick2:=[[3209.153,20.209,-7133.923],[0.5,-0.5,0.5,-0.5],[0,1,-2,0],[500,9E+09,9E+09,9E+09,9E+09,9E+09]];
    CONST robtarget pStackPick2_App:=[[2709.153,20.209,-7133.923],[0.5,-0.5,0.5,-0.5],[0,1,-2,0],[500,9E+09,9E+09,9E+09,9E+09,9E+09]];
    CONST robtarget pStackPlace_App:=[[2262.5,1947.5,610],[0.707106781,0,0,-0.707106781],[0,1,-2,0],[6500,9E+09,9E+09,9E+09,9E+09,9E+09]];
    CONST robtarget pStackPlace:=[[2262.5,1447.5,610],[0.707106781,0,0,-0.707106781],[0,0,-1,0],[6500,9E+09,9E+09,9E+09,9E+09,9E+09]];
    CONST robtarget pStackPlace_Dep_1:=[[2262.5,1247.5,610],[0.707106781,0,0,-0.707106781],[0,0,-1,0],[6500,9E+09,9E+09,9E+09,9E+09,9E+09]];
    CONST robtarget pStackPlace_Dep_2:=[[2262.5,1247.5,-390],[0.707106781,0,0,-0.707106781],[0,0,-1,0],[6500,9E+09,9E+09,9E+09,9E+09,9E+09]];
    !***********************************************************
    !
    ! Module:  Module1
    !
    ! Description:
    !   <Insert description here>
    !
    ! Author: DELL
    !
    ! Version: 1.0
    !
    !***********************************************************


    !***********************************************************
    !
    ! Procedure main
    !
    !   This is the entry point of your program
    !
    !***********************************************************
    PROC main()
        Reset doFeedWheel_L;
        Reset doFeedLink_L;
        Reset doFeedStack;
        Reset doFeedScrews_L;
        Reset doFeedCowCatcher;
        Reset doWheelTool_L;
        Reset doWheel_L;
        Reset doAxel_L;
        Reset doAxelTool_L;
        Reset doLinkTool_L;
        Reset doLink_L;
        Reset doArmTool_L;
        Reset doArm_L;
        Reset doStackTool_L;
        Reset doStack_L;

        SetDO doFeedWheel_L,1;
        SetDO doFeedLink_L, 1;
        SetDO doFeedStack, 1;
        SetDO doFeedScrews_L, 1;

        WHILE TRUE DO
            Reset doFeedWheel_L;
            Reset doFeedLink_L;
            Reset doFeedStack;
            Reset doFeedScrews_L;
            Reset doFeedCowCatcher;
            Reset doWheelTool_L;
            Reset doWheel_L;
            Reset doAxel_L;
            Reset doAxelTool_L;
            Reset doLinkTool_L;
            Reset doLink_L;
            Reset doArmTool_L;
            Reset doArm_L;
            Reset doStackTool_L;
            Reset doStack_L;

            Wheel;
            Axel;
            Link;
            Arm;
            Stack;
        ENDWHILE
    ENDPROC

    PROC Wheel()
        MoveJ pWheel_Home,v1000,z100,tool0\WObj:=Workobject_L;
        MoveJ pWheelTool_App,v1000,fine,tool0\WObj:=Workobject_L;
        MoveL pWheelTool,v500,fine,tool0\WObj:=Workobject_L;
        SetDO doWheelTool_L,1;
        WaitTime 1;
        MoveL pWheelTool_App,v500,fine,WheelTool\WObj:=Workobject_L;
        MoveJ pWheelPick_App,v1000,fine,WheelTool\WObj:=Workobject_L;
        MoveL pWheelPick,v500,fine,WheelTool\WObj:=Workobject_L;
        SetDO doWheel_L,1;
        Reset doFeedWheel_L;
        SetDO doFeedWheel_L,1;
        WaitTime 1;
        MoveL pWheelPick_App,v500,fine,WheelTool\WObj:=Workobject_L;
        MoveJ pWheelPlace1_App,v1000,fine,WheelTool\WObj:=Workobject_L;
        MoveL pWheelPlace1,v200,fine,WheelTool\WObj:=Workobject_L;
        SetDO doWheel_L,0;
        WaitTime 1;
        MoveL pWheelPlace1_App,v200,fine,WheelTool\WObj:=Workobject_L;
        MoveJ pWheelPick_App,v1000,fine,WheelTool\WObj:=Workobject_L;
        MoveL pWheelPick,v500,fine,WheelTool\WObj:=Workobject_L;
        SetDO doWheel_L,1;
        Reset doFeedWheel_L;
        SetDO doFeedWheel_L,1;
        WaitTime 1;
        MoveL pWheelPick_App,v500,fine,WheelTool\WObj:=Workobject_L;
        MoveJ pWheelPlace2_App,v1000,fine,WheelTool\WObj:=Workobject_L;
        MoveL pWheelPlace2,v200,fine,WheelTool\WObj:=Workobject_L;
        SetDO doWheel_L,0;
        WaitTime 1;
        MoveL pWheelPlace2_App,v200,fine,WheelTool\WObj:=Workobject_L;
        MoveJ pWheelTool_App,v1000,fine,WheelTool\WObj:=Workobject_L;
        MoveL pWheelTool,v1000,fine,tool0\WObj:=Workobject_L;
        SetDO doWheelTool_L,0;
        WaitTime 1;
        MoveL pWheelTool_App,v1000,fine,tool0\WObj:=Workobject_L;
        MoveJ pWheel_Home,v1000,z100,tool0\WObj:=Workobject_L;
    ENDPROC

    PROC Axel()
        MoveJ pAxel_Home,v1000,z100,tool0\WObj:=Workobject_L;
        MoveJ pAxelTool_App,v1000,fine,tool0\WObj:=Workobject_L;
        MoveL pAxelTool,v500,fine,tool0\WObj:=Workobject_L;
        SetDO doAxelTool_L,1;
        WaitTime 1;
        MoveL pAxelTool_App,v500,fine,tool0\WObj:=Workobject_L;
        MoveJ pAxelPick1_App,v1000,fine,AxelPinTool\WObj:=Workobject_L;
        MoveL pAxelPick1,v500,fine,AxelPinTool\WObj:=Workobject_L;
        SetDO doAxel_L,1;
        WaitTime 1;
        MoveL pAxelPick1_App,v500,fine,AxelPinTool\WObj:=Workobject_L;
        MoveJ pAxelPlace1_App,v1000,fine,AxelPinTool\WObj:=Workobject_L;
        MoveL pAxelPlace1,v200,fine,AxelPinTool\WObj:=Workobject_L;
        SetDO doAxel_L,0;
        WaitTime 1;
        MoveL pAxelPlace1_App,v200,fine,AxelPinTool\WObj:=Workobject_L;
        MoveJ pAxelPick2_App,v1000,fine,AxelPinTool\WObj:=Workobject_L;
        MoveL pAxelPick2,v500,fine,AxelPinTool\WObj:=Workobject_L;
        SetDO doAxel_L,1;
        WaitTime 1;
        MoveL pAxelPick2_App,v500,fine,AxelPinTool\WObj:=Workobject_L;
        MoveJ pAxelPlace2_App,v1000,fine,AxelPinTool\WObj:=Workobject_L;
        MoveL pAxelPlace2,v200,fine,AxelPinTool\WObj:=Workobject_L;
        SetDO doAxel_L,0;
        WaitTime 1;
        MoveL pAxelPlace2_App,v200,fine,AxelPinTool\WObj:=Workobject_L;
        MoveJ pAxelTool_App,v1000,fine,tool0\WObj:=Workobject_L;
        MoveL pAxelTool,v500,fine,tool0\WObj:=Workobject_L;
        SetDO doAxelTool_L,0;
        WaitTime 1;
        MoveL pAxelTool_App,v500,fine,tool0\WObj:=Workobject_L;
        MoveJ pAxel_Home,v1000,z100,tool0\WObj:=Workobject_L;
    ENDPROC

    PROC Link()
        MoveJ pLink_Home,v1000,z100,tool0\WObj:=Workobject_L;
        MoveJ pLinkTool_App,v1000,fine,tool0\WObj:=Workobject_L;
        MoveL pLinkTool,v500,fine,tool0\WObj:=Workobject_L;
        SetDO doLinkTool_L,1;
        WaitTime 1;
        MoveL pLinkTool_App,v500,fine,tool0\WObj:=Workobject_L;
        MoveJ pLinkPick_App,v1000,fine,LinkTool\WObj:=Workobject_L;
        MoveL pLinkPick,v500,fine,LinkTool\WObj:=Workobject_L;
        SetDO doLink_L,1;
        WaitTime 1;
        MoveL pLinkPick_App,v500,fine,LinkTool\WObj:=Workobject_L;
        MoveJ pLinkPlace_App,v1000,z100,LinkTool\WObj:=Workobject_L;
        MoveL pLinkPlace,v200,fine,LinkTool\WObj:=Workobject_L;
        SetDO doLink_L,0;
        Reset doFeedLink_L;
        SetDO doFeedLink_L,1;
        WaitTime 1;
        MoveL pLinkPlace_App,v200,fine,LinkTool\WObj:=Workobject_L;
        MoveJ pLinkTool_App,v1000,fine,tool0\WObj:=Workobject_L;
        MoveL pLinkTool,v500,fine,tool0\WObj:=Workobject_L;
        SetDO doLinkTool_L,0;
        WaitTime 1;
        MoveL pLinkTool_App,v500,fine,tool0\WObj:=Workobject_L;
        MoveJ pLink_Home,v1000,z100,tool0\WObj:=Workobject_L;
    ENDPROC

    PROC Arm()
        MoveJ pArm_Home,v1000,z100,tool0\WObj:=Workobject_L;
        MoveJ pArmTool_App,v1000,fine,tool0\WObj:=Workobject_L;
        MoveL pArmTool,v500,fine,tool0\WObj:=Workobject_L;
        SetDO doArmTool_L,1;
        WaitTime 1;
        MoveL pArmTool_App,v500,fine,tool0\WObj:=Workobject_L;
        MoveJ pArmPick_App,v1000,fine,ArmPinTool\WObj:=Workobject_L;
        MoveL pArmPick1,v500,fine,ArmPinTool\WObj:=Workobject_L;
        SetDO doArm_L,1;
        WaitTime 1;
        MoveL pArmPick_App,v500,fine,ArmPinTool\WObj:=Workobject_L;
        MoveJ pArmPlace1_App,v1000,fine,ArmPinTool\WObj:=Workobject_L;
        MoveL pArmPlace1,v200,fine,ArmPinTool\WObj:=Workobject_L;
        SetDO doArm_L,0;
        WaitTime 1;
        MoveL pArmPlace1_App,v200,fine,ArmPinTool\WObj:=Workobject_L;
        MoveJ pArmPick_App,v1000,fine,ArmPinTool\WObj:=Workobject_L;
        MoveL pArmPick2,v500,fine,ArmPinTool\WObj:=Workobject_L;
        SetDO doArm_L,1;
        WaitTime 1;
        MoveL pArmPick_App,v500,fine,ArmPinTool\WObj:=Workobject_L;
        MoveJ pArmPlace2_App,v1000,fine,ArmPinTool\WObj:=Workobject_L;
        MoveL pArmPlace2,v500,fine,ArmPinTool\WObj:=Workobject_L;
        SetDO doArm_L,0;
        Reset doFeedScrews_L;
        SetDO doFeedScrews_L,1;
        WaitTime 1;
        MoveL pArmPlace2_App,v500,fine,ArmPinTool\WObj:=Workobject_L;
        MoveJ pArmTool_App,v1000,fine,tool0\WObj:=Workobject_L;
        MoveL pArmTool,v500,fine,tool0\WObj:=Workobject_L;
        SetDO doArmTool_L,0;
        WaitTime 1;
        MoveL pArmTool_App,v500,fine,tool0\WObj:=Workobject_L;
        MoveJ pArm_Home,v1000,z100,tool0\WObj:=Workobject_L;
    ENDPROC

    PROC Stack()
        MoveJ pStack_Home,v1000,z100,tool0\WObj:=Workobject_L;
        MoveJ pStackTool_App,v1000,fine,tool0\WObj:=Workobject_L;
        MoveL pStackTool,v500,fine,tool0\WObj:=Workobject_L;
        SetDO doStackTool_L,1;
        WaitTime 1;
        MoveL pStackTool_App,v500,fine,tool0\WObj:=Workobject_L;
        MoveJ pStack_Home,v1000,z100,StackTool\WObj:=Workobject_L;
        MoveJ pStackPick1_App,v1000,fine,StackTool\WObj:=Workobject_L;
        MoveL pStackPick1,v500,fine,StackTool\WObj:=Workobject_L;
        MoveL pStackPick2,v500,fine,StackTool\WObj:=Workobject_L;
        SetDO doStack_L,1;
        Reset doFeedStack;
        SetDO doFeedStack,1;
        WaitTime 1;
        MoveL pStackPick2_App,v500,fine,StackTool\WObj:=Workobject_L;
        MoveJ pStackPlace_App,v1000,fine,StackTool\WObj:=Workobject_L;
        MoveL pStackPlace,v200,fine,StackTool\WObj:=Workobject_L;
        SetDO doStack_L,0;
        WaitTime 1;
        MoveL pStackPlace_Dep_1,v200,fine,StackTool\WObj:=Workobject_L;
        MoveL pStackPlace_Dep_2,v200,fine,StackTool\WObj:=Workobject_L;
        MoveJ pStackTool_App,v1000,fine,tool0\WObj:=Workobject_L;
        MoveL pStackTool,v500,fine,tool0\WObj:=Workobject_L;
        SetDO doStackTool_L,0;
        WaitTime 1;
        MoveL pStackTool_App,v500,fine,tool0\WObj:=Workobject_L;
        MoveJ pStack_Home,v1000,z100,tool0\WObj:=Workobject_L;
    ENDPROC
ENDMODULE

--- Controller Data/SimulationProject/SYSPAR/EIO.cfg ---
EIO:CFG_1.0:6:1::
#
INDUSTRIAL_NETWORK:

      -Name "PROFIBUS" -Label "PROFIBUS Controller Network"\
      -CfgPath "HOME/pbus_cfg.bin"
#
PROFIBUS_DEVICE:

      -Name "Board10"
#
EIO_SIGNAL:

      -Name "doFeedCowCatcher" -SignalType "DO" -Device "Board10" -DeviceMap "0"

      -Name "doFeedLink_L" -SignalType "DO" -Device "Board10" -DeviceMap "1"

      -Name "doFeedLink_R" -SignalType "DO" -Device "Board10" -DeviceMap "2"

      -Name "doFeedScrews_L" -SignalType "DO" -Device "Board10" -DeviceMap "3"

      -Name "doFeedScrews_R" -SignalType "DO" -Device "Board10" -DeviceMap "4"

      -Name "doFeedStack" -SignalType "DO" -Device "Board10" -DeviceMap "5"

      -Name "doFeedWheel_L" -SignalType "DO" -Device "Board10" -DeviceMap "6"

      -Name "doFeedWheel_R" -SignalType "DO" -Device "Board10" -DeviceMap "7"

      -Name "doWheel" -SignalType "DO" -Device "Board10" -DeviceMap "8"

      -Name "doWheelTool" -SignalType "DO" -Device "Board10" -DeviceMap "9"

      -Name "doAxelTool" -SignalType "DO" -Device "Board10" -DeviceMap "10"

      -Name "doAxel" -SignalType "DO" -Device "Board10" -DeviceMap "11"

      -Name "doLink" -SignalType "DO" -Device "Board10" -DeviceMap "12"

      -Name "doLinkTool" -SignalType "DO" -Device "Board10" -DeviceMap "13"

      -Name "doArm" -SignalType "DO" -Device "Board10" -DeviceMap "14"

      -Name "doArmTool" -SignalType "DO" -Device "Board10" -DeviceMap "15"

      -Name "doCow" -SignalType "DO" -Device "Board10" -DeviceMap "16"

      -Name "doCowTool" -SignalType "DO" -Device "Board10" -DeviceMap "17"

      -Name "doArm_L" -SignalType "DO" -Device "Board10" -DeviceMap "18"

      -Name "doArmTool_L" -SignalType "DO" -Device "Board10" -DeviceMap "19"

      -Name "doAxel_L" -SignalType "DO" -Device "Board10" -DeviceMap "20"

      -Name "doAxelTool_L" -SignalType "DO" -Device "Board10" -DeviceMap "21"

      -Name "doStack_L" -SignalType "DO" -Device "Board10" -DeviceMap "22"

      -Name "doStackTool_L" -SignalType "DO" -Device "Board10" -DeviceMap "23"

      -Name "doLink_L" -SignalType "DO" -Device "Board10" -DeviceMap "24"

      -Name "doLinkTool_L" -SignalType "DO" -Device "Board10" -DeviceMap "25"

      -Name "doWheel_L" -SignalType "DO" -Device "Board10" -DeviceMap "26"

      -Name "doWheelTool_L" -SignalType "DO" -Device "Board10" -DeviceMap "27"
